LIN {X 0,Y 288.078,Z 352.641,A -85,B 0,C 180,E1 -18480.944,E2 -18480.944} C_VEL
LIN {X 0,Y 287.498,Z 347.512,A -85,B 0,C 180,E1 -18481.625,E2 -18481.625} C_VEL
LIN {X 0,Y 284.939,Z 340.607,A -85,B 0,C 180,E1 -18483.326,E2 -18483.326} C_VEL
LIN {X 0,Y 282.556,Z 335.313,A -85,B 0,C 180,E1 -18485.033,E2 -18485.033} C_VEL
LIN {X 0,Y 279.888,Z 329.784,A -85,B 0,C 180,E1 -18487.357,E2 -18487.357} C_VEL
LIN {X 0,Y 277.601,Z 325.434,A -85,B 0,C 180,E1 -18490.071,E2 -18490.071} C_VEL
LIN {X 0,Y 276.504,Z 323.001,A -85,B 0,C 180,E1 -18492.267,E2 -18492.267} C_VEL
LIN {X 0,Y 275.913,Z 321.671,A -85,B 0,C 180,E1 -18494.976,E2 -18494.976} C_VEL
LIN {X 0,Y 276.373,Z 321.734,A -85,B 0,C 180,E1 -18497.824,E2 -18497.824} C_VEL
LIN {X 0,Y 278.265,Z 323.737,A -85,B 0,C 180,E1 -18501.065,E2 -18501.065} C_VEL
LIN {X 0,Y 279.613,Z 325.391,A -85,B 0,C 180,E1 -18502.576,E2 -18502.576} C_VEL
LIN {X 0,Y 282.459,Z 329.547,A -85,B 0,C 180,E1 -18505.038,E2 -18505.038} C_VEL
LIN {X 0,Y 285.243,Z 334.015,A -85,B 0,C 180,E1 -18506.959,E2 -18506.959} C_VEL
LIN {X 0,Y 288.63,Z 340.16,A -85,B 0,C 180,E1 -18508.952,E2 -18508.952} C_VEL
LIN {X 0,Y 290.717,Z 344.56,A -85,B 0,C 180,E1 -18510.068,E2 -18510.068} C_VEL
LIN {X 0,Y 285.573,Z 380.843,A -85,B 0,C 180,E1 -18511.832,E2 -18511.832} C_VEL
LIN {X 0,Y 283.258,Z 392.365,A -85,B 0,C 180,E1 -18512.67,E2 -18512.67} C_VEL
LIN {X 0,Y 280.814,Z 402.262,A -85,B 0,C 180,E1 -18513.619,E2 -18513.619} C_VEL
LIN {X 0,Y 277.418,Z 413.784,A -85,B 0,C 180,E1 -18515.085,E2 -18515.085} C_VEL
LIN {X 0,Y 274.94,Z 421.064,A -85,B 0,C 180,E1 -18516.253,E2 -18516.253} C_VEL
LIN {X 0,Y 272.241,Z 428.033,A -85,B 0,C 180,E1 -18517.612,E2 -18517.612} C_VEL
LIN {X 0,Y 269.739,Z 433.852,A -85,B 0,C 180,E1 -18519,E2 -18519} C_VEL
LIN {X 0,Y 266.409,Z 441.005,A -85,B 0,C 180,E1 -18521.139,E2 -18521.139} C_VEL
LIN {X 0,Y 263.86,Z 445.653,A -85,B 0,C 180,E1 -18522.956,E2 -18522.956} C_VEL
LIN {X 0,Y 261.191,Z 449.803,A -85,B 0,C 180,E1 -18525.182,E2 -18525.182} C_VEL
LIN {X 0,Y 258.896,Z 452.702,A -85,B 0,C 180,E1 -18527.45,E2 -18527.45} C_VEL
LIN {X 0,Y 257.809,Z 453.984,A -85,B 0,C 180,E1 -18528.992,E2 -18528.992} C_VEL
LIN {X 0,Y 256.643,Z 454.794,A -85,B 0,C 180,E1 -18530.536,E2 -18530.536} C_VEL
LIN {X 0,Y 255.749,Z 454.994,A -85,B 0,C 180,E1 -18532.095,E2 -18532.095} C_VEL
LIN {X 0,Y 255.162,Z 454.673,A -85,B 0,C 180,E1 -18533.667,E2 -18533.667} C_VEL
LIN {X 0,Y 254.747,Z 453.89,A -85,B 0,C 180,E1 -18535.245,E2 -18535.245} C_VEL
LIN {X 0,Y 254.42,Z 452.619,A -85,B 0,C 180,E1 -18536.825,E2 -18536.825} C_VEL
LIN {X 0,Y 254.109,Z 449.575,A -85,B 0,C 180,E1 -18539.2,E2 -18539.2} C_VEL
LIN {X 0,Y 254.108,Z 445.253,A -85,B 0,C 180,E1 -18541.577,E2 -18541.577} C_VEL
LIN {X 0,Y 254.373,Z 439.511,A -85,B 0,C 180,E1 -18543.952,E2 -18543.952} C_VEL
LIN {X 0,Y 254.476,Z 433.189,A -85,B 0,C 180,E1 -18545.929,E2 -18545.929} C_VEL
LIN {X 0,Y 254.903,Z 425.839,A -85,B 0,C 180,E1 -18547.78,E2 -18547.78} C_VEL
LIN {X 0,Y 255.323,Z 417.479,A -85,B 0,C 180,E1 -18549.498,E2 -18549.498} C_VEL
LIN {X 0,Y 255.884,Z 406.564,A -85,B 0,C 180,E1 -18551.276,E2 -18551.276} C_VEL
LIN {X 0,Y 256.338,Z 397.268,A -85,B 0,C 180,E1 -18552.46,E2 -18552.46} C_VEL
LIN {X 0,Y 256.889,Z 386.565,A -85,B 0,C 180,E1 -18553.539,E2 -18553.539} C_VEL
LIN {X 0,Y 257.314,Z 373.603,A -85,B 0,C 180,E1 -18554.474,E2 -18554.474} C_VEL
LIN {X 0,Y 258.64,Z 317.417,A -85,B 0,C 180,E1 -18557.079,E2 -18557.079} C_VEL
LIN {X 0,Y 256.336,Z 296.461,A -85,B 0,C 180,E1 -18558.059,E2 -18558.059} C_VEL
LIN {X 0,Y 256.227,Z 294.598,A -85,B 0,C 180,E1 -18558.171,E2 -18558.171} C_VEL
LIN {X 0,Y 256.274,Z 293.374,A -85,B 0,C 180,E1 -18558.788,E2 -18558.788} C_VEL
LIN {X 0,Y 256.19,Z 293.381,A -85,B 0,C 180,E1 -18561.133,E2 -18561.133} C_VEL
LIN {X 0,Y 256.054,Z 293.402,A -85,B 0,C 180,E1 -18566.04,E2 -18566.04} C_VEL
LIN {X 0,Y 256.026,Z 293.403,A -85,B 0,C 180,E1 -18569.6,E2 -18569.6} C_VEL
LIN {X 0,Y 256.048,Z 293.399,A -85,B 0,C 180,E1 -18573.284,E2 -18573.284} C_VEL
LIN {X 0,Y 256.066,Z 293.398,A -85,B 0,C 180,E1 -18577.253,E2 -18577.253} C_VEL
LIN {X 0,Y 255.984,Z 293.408,A -85,B 0,C 180,E1 -18581.204,E2 -18581.204} C_VEL
LIN {X 0,Y 256.009,Z 293.405,A -85,B 0,C 180,E1 -18585.527,E2 -18585.527} C_VEL
LIN {X 0,Y 256.021,Z 293.406,A -85,B 0,C 180,E1 -18588.787,E2 -18588.787} C_VEL
LIN {X 0,Y 256.097,Z 293.398,A -85,B 0,C 180,E1 -18592.859,E2 -18592.859} C_VEL
LIN {X 0,Y 256.031,Z 293.404,A -85,B 0,C 180,E1 -18596.699,E2 -18596.699} C_VEL
LIN {X 0,Y 256.028,Z 293.402,A -85,B 0,C 180,E1 -18600.387,E2 -18600.387} C_VEL
LIN {X 0,Y 256.088,Z 293.396,A -85,B 0,C 180,E1 -18603.951,E2 -18603.951} C_VEL
LIN {X 0,Y 256.041,Z 293.403,A -85,B 0,C 180,E1 -18607.398,E2 -18607.398} C_VEL
LIN {X 0,Y 256.14,Z 293.389,A -85,B 0,C 180,E1 -18610.774,E2 -18610.774} C_VEL
LIN {X 0,Y 256.22,Z 293.379,A -85,B 0,C 180,E1 -18614.077,E2 -18614.077} C_VEL
LIN {X 0,Y 256.262,Z 293.373,A -85,B 0,C 180,E1 -18618.929,E2 -18618.929} C_VEL
LIN {X 0,Y 256.482,Z 293.348,A -85,B 0,C 180,E1 -18622.123,E2 -18622.123} C_VEL
LIN {X 0,Y 256.672,Z 293.324,A -85,B 0,C 180,E1 -18628.428,E2 -18628.428} C_VEL
LIN {X 0,Y 256.671,Z 293.324,A -85,B 0,C 180,E1 -18631.566,E2 -18631.566} C_VEL
LIN {X 0,Y 256.478,Z 293.349,A -85,B 0,C 180,E1 -18637.872,E2 -18637.872} C_VEL
LIN {X 0,Y 256.258,Z 293.374,A -85,B 0,C 180,E1 -18641.065,E2 -18641.065} C_VEL
LIN {X 0,Y 256.213,Z 293.38,A -85,B 0,C 180,E1 -18645.917,E2 -18645.917} C_VEL
LIN {X 0,Y 256.132,Z 293.39,A -85,B 0,C 180,E1 -18649.221,E2 -18649.221} C_VEL
LIN {X 0,Y 256.032,Z 293.404,A -85,B 0,C 180,E1 -18652.597,E2 -18652.597} C_VEL
LIN {X 0,Y 256.079,Z 293.397,A -85,B 0,C 180,E1 -18656.044,E2 -18656.044} C_VEL
LIN {X 0,Y 256.065,Z 293.397,A -85,B 0,C 180,E1 -18659.602,E2 -18659.602} C_VEL
LIN {X 0,Y 256.038,Z 293.403,A -85,B 0,C 180,E1 -18663.293,E2 -18663.293} C_VEL
LIN {X 0,Y 256.093,Z 293.397,A -85,B 0,C 180,E1 -18667.282,E2 -18667.282} C_VEL
LIN {X 0,Y 256.088,Z 293.398,A -85,B 0,C 180,E1 -18671.193,E2 -18671.193} C_VEL
LIN {X 0,Y 256.074,Z 293.4,A -85,B 0,C 180,E1 -18675.522,E2 -18675.522} C_VEL
LIN {X 0,Y 256.091,Z 293.395,A -85,B 0,C 180,E1 -18678.817,E2 -18678.817} C_VEL
LIN {X 0,Y 256.115,Z 293.392,A -85,B 0,C 180,E1 -18682.877,E2 -18682.877} C_VEL
LIN {X 0,Y 256.049,Z 293.399,A -85,B 0,C 180,E1 -18686.716,E2 -18686.716} C_VEL
LIN {X 0,Y 256.093,Z 293.397,A -85,B 0,C 180,E1 -18691.417,E2 -18691.417} C_VEL
LIN {X 0,Y 256.111,Z 293.396,A -85,B 0,C 180,E1 -18695.704,E2 -18695.704} C_VEL
LIN {X 0,Y 256.119,Z 293.39,A -85,B 0,C 180,E1 -18699.111,E2 -18699.111} C_VEL
LIN {X 0,Y 256.22,Z 293.382,A -85,B 0,C 180,E1 -18704.089,E2 -18704.089} C_VEL
LIN {X 0,Y 256.268,Z 293.373,A -85,B 0,C 180,E1 -18708.941,E2 -18708.941} C_VEL
LIN {X 0,Y 256.478,Z 293.351,A -85,B 0,C 180,E1 -18712.134,E2 -18712.134} C_VEL
LIN {X 0,Y 256.439,Z 293.352,A -85,B 0,C 180,E1 -18716.866,E2 -18716.866} C_VEL
LIN {X 0,Y 256.686,Z 293.325,A -85,B 0,C 180,E1 -18718.439,E2 -18718.439} C_VEL
LIN {X 0,Y 256.686,Z 293.321,A -85,B 0,C 180,E1 -18721.577,E2 -18721.577} C_VEL
LIN {X 0,Y 256.445,Z 293.351,A -85,B 0,C 180,E1 -18726.301,E2 -18726.301} C_VEL
LIN {X 0,Y 256.393,Z 293.358,A -85,B 0,C 180,E1 -18729.474,E2 -18729.474} C_VEL
LIN {X 0,Y 256.198,Z 293.38,A -85,B 0,C 180,E1 -18734.301,E2 -18734.301} C_VEL
LIN {X 0,Y 256.142,Z 293.389,A -85,B 0,C 180,E1 -18737.574,E2 -18737.574} C_VEL
LIN {X 0,Y 256.115,Z 293.395,A -85,B 0,C 180,E1 -18741.104,E2 -18741.104} C_VEL
LIN {X 0,Y 256.083,Z 293.399,A -85,B 0,C 180,E1 -18745.096,E2 -18745.096} C_VEL
LIN {X 0,Y 256.086,Z 293.396,A -85,B 0,C 180,E1 -18748.581,E2 -18748.581} C_VEL
LIN {X 0,Y 256.075,Z 293.398,A -85,B 0,C 180,E1 -18751.708,E2 -18751.708} C_VEL
LIN {X 0,Y 256.066,Z 293.399,A -85,B 0,C 180,E1 -18753.482,E2 -18753.482} C_VEL
LIN {X 0,Y 255.413,Z 293.481,A -85,B 0,C 180,E1 -18754.795,E2 -18754.795} C_VEL
LIN {X 0,Y 252.605,Z 293.833,A -85,B 0,C 180,E1 -18756.938,E2 -18756.938} C_VEL
LIN {X 0,Y 249.35,Z 294.238,A -85,B 0,C 180,E1 -18759.577,E2 -18759.577} C_VEL
LIN {X 0,Y 248.983,Z 294.278,A -85,B 0,C 180,E1 -18760.491,E2 -18760.491} C_VEL
LIN {X 0,Y 248.968,Z 294.282,A -85,B 0,C 180,E1 -18764.895,E2 -18764.895} C_VEL
LIN {X 0,Y 248.986,Z 294.281,A -85,B 0,C 180,E1 -18767.361,E2 -18767.361} C_VEL
LIN {X 0,Y 249.053,Z 294.274,A -85,B 0,C 180,E1 -18772.207,E2 -18772.207} C_VEL
LIN {X 0,Y 249.053,Z 294.273,A -85,B 0,C 180,E1 -18775.645,E2 -18775.645} C_VEL
LIN {X 0,Y 249.01,Z 294.275,A -85,B 0,C 180,E1 -18779.471,E2 -18779.471} C_VEL
LIN {X 0,Y 249.328,Z 294.267,A -85,B 0,C 180,E1 -18783.991,E2 -18783.991} C_VEL
LIN {X 0,Y 250.346,Z 300.279,A -85,B 0,C 180,E1 -18786.423,E2 -18786.423} C_VEL
LIN {X 0,Y 249.092,Z 310.954,A -85,B 0,C 180,E1 -18790.642,E2 -18790.642} C_VEL
LIN {X 0,Y 248.799,Z 313.594,A -85,B 0,C 180,E1 -18791.687,E2 -18791.687} C_VEL
LIN {X 0,Y 249.482,Z 331.264,A -85,B 0,C 180,E1 -18792.554,E2 -18792.554} C_VEL
LIN {X 0,Y 251.209,Z 351.622,A -85,B 0,C 180,E1 -18793.536,E2 -18793.536} C_VEL
LIN {X 0,Y 250.2,Z 393.642,A -85,B 0,C 180,E1 -18795.619,E2 -18795.619} C_VEL
LIN {X 0,Y 249.777,Z 405.976,A -85,B 0,C 180,E1 -18796.58,E2 -18796.58} C_VEL
LIN {X 0,Y 249.294,Z 415.542,A -85,B 0,C 180,E1 -18797.59,E2 -18797.59} C_VEL
LIN {X 0,Y 248.756,Z 426.15,A -85,B 0,C 180,E1 -18799.009,E2 -18799.009} C_VEL
LIN {X 0,Y 248.379,Z 435.573,A -85,B 0,C 180,E1 -18800.639,E2 -18800.639} C_VEL
LIN {X 0,Y 248.049,Z 443.217,A -85,B 0,C 180,E1 -18802.274,E2 -18802.274} C_VEL
LIN {X 0,Y 247.91,Z 449.562,A -85,B 0,C 180,E1 -18803.91,E2 -18803.91} C_VEL
LIN {X 0,Y 247.768,Z 454.731,A -85,B 0,C 180,E1 -18805.529,E2 -18805.529} C_VEL
LIN {X 0,Y 247.6,Z 459.948,A -85,B 0,C 180,E1 -18807.563,E2 -18807.563} C_VEL
LIN {X 0,Y 247.634,Z 464.762,A -85,B 0,C 180,E1 -18810.003,E2 -18810.003} C_VEL
LIN {X 0,Y 247.206,Z 466.989,A -85,B 0,C 180,E1 -18811.632,E2 -18811.632} C_VEL
LIN {X 0,Y 247.115,Z 468.697,A -85,B 0,C 180,E1 -18813.263,E2 -18813.263} C_VEL
LIN {X 0,Y 247.11,Z 470.165,A -85,B 0,C 180,E1 -18815.429,E2 -18815.429} C_VEL
LIN {X 0,Y 247.201,Z 470.623,A -85,B 0,C 180,E1 -18816.533,E2 -18816.533} C_VEL
LIN {X 0,Y 247.539,Z 470.786,A -85,B 0,C 180,E1 -18818.164,E2 -18818.164} C_VEL
LIN {X 0,Y 248.096,Z 470.422,A -85,B 0,C 180,E1 -18819.789,E2 -18819.789} C_VEL
LIN {X 0,Y 248.913,Z 469.615,A -85,B 0,C 180,E1 -18821.402,E2 -18821.402} C_VEL
LIN {X 0,Y 249.993,Z 468.35,A -85,B 0,C 180,E1 -18823,E2 -18823} C_VEL
LIN {X 0,Y 252.028,Z 465.39,A -85,B 0,C 180,E1 -18825.364,E2 -18825.364} C_VEL
LIN {X 0,Y 253.723,Z 462.798,A -85,B 0,C 180,E1 -18826.911,E2 -18826.911} C_VEL
LIN {X 0,Y 256.501,Z 457.656,A -85,B 0,C 180,E1 -18829.198,E2 -18829.198} C_VEL
LIN {X 0,Y 259.354,Z 452.305,A -85,B 0,C 180,E1 -18831.044,E2 -18831.044} C_VEL
LIN {X 0,Y 262.607,Z 445.702,A -85,B 0,C 180,E1 -18832.836,E2 -18832.836} C_VEL
LIN {X 0,Y 266.26,Z 437.594,A -85,B 0,C 180,E1 -18834.567,E2 -18834.567} C_VEL
LIN {X 0,Y 269.842,Z 428.59,A -85,B 0,C 180,E1 -18836.075,E2 -18836.075} C_VEL
LIN {X 0,Y 272.91,Z 420.038,A -85,B 0,C 180,E1 -18837.202,E2 -18837.202} C_VEL
LIN {X 0,Y 275.659,Z 411.201,A -85,B 0,C 180,E1 -18838.145,E2 -18838.145} C_VEL
LIN {X 0,Y 278.901,Z 399.082,A -85,B 0,C 180,E1 -18839.123,E2 -18839.123} C_VEL
LIN {X 0,Y 281.328,Z 386.651,A -85,B 0,C 180,E1 -18839.875,E2 -18839.875} C_VEL
LIN {X 0,Y 284.531,Z 364.834,A -85,B 0,C 180,E1 -18840.937,E2 -18840.937} C_VEL
LIN {X 0,Y 284.092,Z 354.378,A -85,B 0,C 180,E1 -18842.129,E2 -18842.129} C_VEL
LIN {X 0,Y 283.77,Z 351.646,A -85,B 0,C 180,E1 -18842.551,E2 -18842.551} C_VEL
LIN {X 0,Y 281.525,Z 345.515,A -85,B 0,C 180,E1 -18844.168,E2 -18844.168} C_VEL
LIN {X 0,Y 279.677,Z 341.044,A -85,B 0,C 180,E1 -18845.691,E2 -18845.691} C_VEL
LIN {X 0,Y 277.489,Z 336.114,A -85,B 0,C 180,E1 -18847.818,E2 -18847.818} C_VEL
LIN {X 0,Y 275.344,Z 331.685,A -85,B 0,C 180,E1 -18850.66,E2 -18850.66} C_VEL
LIN {X 0,Y 274.535,Z 329.607,A -85,B 0,C 180,E1 -18852.644,E2 -18852.644} C_VEL
LIN {X 0,Y 274.11,Z 328.543,A -85,B 0,C 180,E1 -18854.977,E2 -18854.977} C_VEL
LIN {X 0,Y 274.456,Z 328.463,A -85,B 0,C 180,E1 -18857.484,E2 -18857.484} C_VEL
LIN {X 0,Y 276.365,Z 330.545,A -85,B 0,C 180,E1 -18860.979,E2 -18860.979} C_VEL
LIN {X 0,Y 277.561,Z 332.177,A -85,B 0,C 180,E1 -18862.414,E2 -18862.414} C_VEL
LIN {X 0,Y 279.95,Z 335.855,A -85,B 0,C 180,E1 -18864.624,E2 -18864.624} C_VEL
LIN {X 0,Y 282.575,Z 340.41,A -85,B 0,C 180,E1 -18866.592,E2 -18866.592} C_VEL
LIN {X 0,Y 285.617,Z 346.256,A -85,B 0,C 180,E1 -18868.504,E2 -18868.504} C_VEL
LIN {X 0,Y 286.579,Z 348.295,A -85,B 0,C 180,E1 -18869.052,E2 -18869.052} C_VEL
LIN {X 0,Y 281.589,Z 380.533,A -85,B 0,C 180,E1 -18870.614,E2 -18870.614} C_VEL
LIN {X 0,Y 279.233,Z 391.744,A -85,B 0,C 180,E1 -18871.425,E2 -18871.425} C_VEL
LIN {X 0,Y 276.604,Z 401.83,A -85,B 0,C 180,E1 -18872.367,E2 -18872.367} C_VEL
LIN {X 0,Y 273.406,Z 412.453,A -85,B 0,C 180,E1 -18873.671,E2 -18873.671} C_VEL
LIN {X 0,Y 270.319,Z 420.838,A -85,B 0,C 180,E1 -18875.002,E2 -18875.002} C_VEL
LIN {X 0,Y 266.726,Z 429.403,A -85,B 0,C 180,E1 -18876.712,E2 -18876.712} C_VEL
LIN {X 0,Y 263.432,Z 436.434,A -85,B 0,C 180,E1 -18878.473,E2 -18878.473} C_VEL
LIN {X 0,Y 260.508,Z 442,A -85,B 0,C 180,E1 -18880.285,E2 -18880.285} C_VEL
LIN {X 0,Y 257.237,Z 447.173,A -85,B 0,C 180,E1 -18882.503,E2 -18882.503} C_VEL
LIN {X 0,Y 254.456,Z 451.035,A -85,B 0,C 180,E1 -18884.781,E2 -18884.781} C_VEL
LIN {X 0,Y 253.559,Z 452.117,A -85,B 0,C 180,E1 -18885.547,E2 -18885.547} C_VEL
LIN {X 0,Y 252.043,Z 453.653,A -85,B 0,C 180,E1 -18887.103,E2 -18887.103} C_VEL
LIN {X 0,Y 250.885,Z 454.66,A -85,B 0,C 180,E1 -18888.684,E2 -18888.684} C_VEL
LIN {X 0,Y 249.669,Z 455.239,A -85,B 0,C 180,E1 -18890.269,E2 -18890.269} C_VEL
LIN {X 0,Y 248.732,Z 455.338,A -85,B 0,C 180,E1 -18891.871,E2 -18891.871} C_VEL
LIN {X 0,Y 248.107,Z 454.848,A -85,B 0,C 180,E1 -18893.486,E2 -18893.486} C_VEL
LIN {X 0,Y 247.682,Z 453.826,A -85,B 0,C 180,E1 -18895.109,E2 -18895.109} C_VEL
LIN {X 0,Y 247.211,Z 451.421,A -85,B 0,C 180,E1 -18897.548,E2 -18897.548} C_VEL
LIN {X 0,Y 247.02,Z 447.737,A -85,B 0,C 180,E1 -18899.992,E2 -18899.992} C_VEL
LIN {X 0,Y 247.135,Z 442.542,A -85,B 0,C 180,E1 -18902.436,E2 -18902.436} C_VEL
LIN {X 0,Y 247.322,Z 438.239,A -85,B 0,C 180,E1 -18904.065,E2 -18904.065} C_VEL
LIN {X 0,Y 247.471,Z 431.905,A -85,B 0,C 180,E1 -18906.014,E2 -18906.014} C_VEL
LIN {X 0,Y 247.853,Z 425.134,A -85,B 0,C 180,E1 -18907.732,E2 -18907.732} C_VEL
LIN {X 0,Y 248.308,Z 416.296,A -85,B 0,C 180,E1 -18909.563,E2 -18909.563} C_VEL
LIN {X 0,Y 248.805,Z 406.247,A -85,B 0,C 180,E1 -18911.189,E2 -18911.189} C_VEL
LIN {X 0,Y 249.261,Z 396.831,A -85,B 0,C 180,E1 -18912.406,E2 -18912.406} C_VEL
LIN {X 0,Y 249.824,Z 385.992,A -85,B 0,C 180,E1 -18913.514,E2 -18913.514} C_VEL
LIN {X 0,Y 250.222,Z 373.37,A -85,B 0,C 180,E1 -18914.425,E2 -18914.425} C_VEL
LIN {X 0,Y 251.46,Z 317.095,A -85,B 0,C 180,E1 -18917.152,E2 -18917.152} C_VEL
LIN {X 0,Y 249.248,Z 296.678,A -85,B 0,C 180,E1 -18918.139,E2 -18918.139} C_VEL
LIN {X 0,Y 249.146,Z 294.806,A -85,B 0,C 180,E1 -18918.28,E2 -18918.28} C_VEL
LIN {X 0,Y 249.181,Z 294.258,A -85,B 0,C 180,E1 -18918.597,E2 -18918.597} C_VEL
LIN {X 0,Y 249.097,Z 294.266,A -85,B 0,C 180,E1 -18921.507,E2 -18921.507} C_VEL
LIN {X 0,Y 249.033,Z 294.274,A -85,B 0,C 180,E1 -18925.43,E2 -18925.43} C_VEL
LIN {X 0,Y 249.01,Z 294.277,A -85,B 0,C 180,E1 -18928.958,E2 -18928.958} C_VEL
LIN {X 0,Y 249.009,Z 294.279,A -85,B 0,C 180,E1 -18932.417,E2 -18932.417} C_VEL
LIN {X 0,Y 248.991,Z 294.283,A -85,B 0,C 180,E1 -18936.339,E2 -18936.339} C_VEL
LIN {X 0,Y 248.949,Z 294.286,A -85,B 0,C 180,E1 -18940.476,E2 -18940.476} C_VEL
LIN {X 0,Y 248.948,Z 294.288,A -85,B 0,C 180,E1 -18944.877,E2 -18944.877} C_VEL
LIN {X 0,Y 248.978,Z 294.281,A -85,B 0,C 180,E1 -18947.352,E2 -18947.352} C_VEL
LIN {X 0,Y 249.011,Z 294.277,A -85,B 0,C 180,E1 -18952.192,E2 -18952.192} C_VEL
LIN {X 0,Y 249.009,Z 294.277,A -85,B 0,C 180,E1 -18955.631,E2 -18955.631} C_VEL
LIN {X 0,Y 248.97,Z 294.283,A -85,B 0,C 180,E1 -18959.459,E2 -18959.459} C_VEL
LIN {X 0,Y 249.024,Z 294.279,A -85,B 0,C 180,E1 -18963.154,E2 -18963.154} C_VEL
LIN {X 0,Y 249.019,Z 294.275,A -85,B 0,C 180,E1 -18966.724,E2 -18966.724} C_VEL
LIN {X 0,Y 249.064,Z 294.27,A -85,B 0,C 180,E1 -18970.205,E2 -18970.205} C_VEL
LIN {X 0,Y 249.152,Z 294.263,A -85,B 0,C 180,E1 -18973.613,E2 -18973.613} C_VEL
LIN {X 0,Y 249.205,Z 294.252,A -85,B 0,C 180,E1 -18978.612,E2 -18978.612} C_VEL
LIN {X 0,Y 249.423,Z 294.229,A -85,B 0,C 180,E1 -18981.898,E2 -18981.898} C_VEL
LIN {X 0,Y 249.416,Z 294.225,A -85,B 0,C 180,E1 -18986.767,E2 -18986.767} C_VEL
LIN {X 0,Y 249.685,Z 294.198,A -85,B 0,C 180,E1 -18989.997,E2 -18989.997} C_VEL
LIN {X 0,Y 249.414,Z 294.225,A -85,B 0,C 180,E1 -18993.228,E2 -18993.228} C_VEL
LIN {X 0,Y 249.419,Z 294.229,A -85,B 0,C 180,E1 -18998.096,E2 -18998.096} C_VEL
LIN {X 0,Y 249.2,Z 294.253,A -85,B 0,C 180,E1 -19001.383,E2 -19001.383} C_VEL
LIN {X 0,Y 249.146,Z 294.264,A -85,B 0,C 180,E1 -19006.486,E2 -19006.486} C_VEL
LIN {X 0,Y 249.043,Z 294.271,A -85,B 0,C 180,E1 -19011.399,E2 -19011.399} C_VEL
LIN {X 0,Y 249.067,Z 294.27,A -85,B 0,C 180,E1 -19015.477,E2 -19015.477} C_VEL
LIN {X 0,Y 249.034,Z 294.276,A -85,B 0,C 180,E1 -19018.995,E2 -19018.995} C_VEL
LIN {X 0,Y 248.988,Z 294.279,A -85,B 0,C 180,E1 -19022.428,E2 -19022.428} C_VEL
LIN {X 0,Y 249.028,Z 294.275,A -85,B 0,C 180,E1 -19026.342,E2 -19026.342} C_VEL
LIN {X 0,Y 249.039,Z 294.271,A -85,B 0,C 180,E1 -19030.467,E2 -19030.467} C_VEL
LIN {X 0,Y 249.05,Z 294.273,A -85,B 0,C 180,E1 -19032.818,E2 -19032.818} C_VEL
LIN {X 0,Y 249.057,Z 294.274,A -85,B 0,C 180,E1 -19037.385,E2 -19037.385} C_VEL
LIN {X 0,Y 249.013,Z 294.28,A -85,B 0,C 180,E1 -19041.63,E2 -19041.63} C_VEL
LIN {X 0,Y 249.025,Z 294.278,A -85,B 0,C 180,E1 -19045.649,E2 -19045.649} C_VEL
LIN {X 0,Y 249.013,Z 294.277,A -85,B 0,C 180,E1 -19049.479,E2 -19049.479} C_VEL
LIN {X 0,Y 249.036,Z 294.275,A -85,B 0,C 180,E1 -19053.169,E2 -19053.169} C_VEL
LIN {X 0,Y 249.03,Z 294.272,A -85,B 0,C 180,E1 -19056.738,E2 -19056.738} C_VEL
LIN {X 0,Y 249.054,Z 294.274,A -85,B 0,C 180,E1 -19060.217,E2 -19060.217} C_VEL
LIN {X 0,Y 249.17,Z 294.259,A -85,B 0,C 180,E1 -19063.626,E2 -19063.626} C_VEL
LIN {X 0,Y 249.211,Z 294.253,A -85,B 0,C 180,E1 -19068.624,E2 -19068.624} C_VEL
LIN {X 0,Y 249.421,Z 294.228,A -85,B 0,C 180,E1 -19071.91,E2 -19071.91} C_VEL
LIN {X 0,Y 249.253,Z 294.244,A -85,B 0,C 180,E1 -19075.156,E2 -19075.156} C_VEL
LIN {X 0,Y 249.646,Z 294.201,A -85,B 0,C 180,E1 -19078.395,E2 -19078.395} C_VEL
LIN {X 0,Y 249.647,Z 294.197,A -85,B 0,C 180,E1 -19081.621,E2 -19081.621} C_VEL
LIN {X 0,Y 249.416,Z 294.228,A -85,B 0,C 180,E1 -19086.479,E2 -19086.479} C_VEL
LIN {X 0,Y 249.324,Z 294.238,A -85,B 0,C 180,E1 -19089.745,E2 -19089.745} C_VEL
LIN {X 0,Y 249.142,Z 294.261,A -85,B 0,C 180,E1 -19094.715,E2 -19094.715} C_VEL
LIN {X 0,Y 249.074,Z 294.269,A -85,B 0,C 180,E1 -19098.09,E2 -19098.09} C_VEL
LIN {X 0,Y 249.039,Z 294.272,A -85,B 0,C 180,E1 -19101.53,E2 -19101.53} C_VEL
LIN {X 0,Y 249.045,Z 294.276,A -85,B 0,C 180,E1 -19105.448,E2 -19105.448} C_VEL
LIN {X 0,Y 249.034,Z 294.276,A -85,B 0,C 180,E1 -19108.98,E2 -19108.98} C_VEL
LIN {X 0,Y 249.003,Z 294.273,A -85,B 0,C 180,E1 -19113.487,E2 -19113.487} C_VEL
LIN {X 0,Y 249.047,Z 294.274,A -85,B 0,C 180,E1 -19117.806,E2 -19117.806} C_VEL
LIN {X 0,Y 248.983,Z 294.278,A -85,B 0,C 180,E1 -19120.491,E2 -19120.491} C_VEL
LIN {X 0,Y 248.239,Z 294.376,A -85,B 0,C 180,E1 -19121.84,E2 -19121.84} C_VEL
LIN {X 0,Y 245.348,Z 294.736,A -85,B 0,C 180,E1 -19124.04,E2 -19124.04} C_VEL
LIN {X 0,Y 242.957,Z 295.035,A -85,B 0,C 180,E1 -19125.832,E2 -19125.832} C_VEL
LIN {X 0,Y 241.963,Z 295.155,A -85,B 0,C 180,E1 -19127.221,E2 -19127.221} C_VEL
LIN {X 0,Y 241.897,Z 295.161,A -85,B 0,C 180,E1 -19127.692,E2 -19127.692} C_VEL
LIN {X 0,Y 242.003,Z 295.151,A -85,B 0,C 180,E1 -19131.648,E2 -19131.648} C_VEL
LIN {X 0,Y 241.984,Z 295.154,A -85,B 0,C 180,E1 -19134.493,E2 -19134.493} C_VEL
LIN {X 0,Y 241.961,Z 295.155,A -85,B 0,C 180,E1 -19138.482,E2 -19138.482} C_VEL
LIN {X 0,Y 242.307,Z 295.12,A -85,B 0,C 180,E1 -19144.135,E2 -19144.135} C_VEL
LIN {X 0,Y 243.237,Z 299.948,A -85,B 0,C 180,E1 -19146.143,E2 -19146.143} C_VEL
LIN {X 0,Y 242.392,Z 307.442,A -85,B 0,C 180,E1 -19149.199,E2 -19149.199} C_VEL
LIN {X 0,Y 241.726,Z 313.336,A -85,B 0,C 180,E1 -19151.613,E2 -19151.613} C_VEL
LIN {X 0,Y 242.353,Z 331.256,A -85,B 0,C 180,E1 -19152.547,E2 -19152.547} C_VEL
LIN {X 0,Y 244.114,Z 351.259,A -85,B 0,C 180,E1 -19153.54,E2 -19153.54} C_VEL
LIN {X 0,Y 243.141,Z 392.775,A -85,B 0,C 180,E1 -19155.674,E2 -19155.674} C_VEL
LIN {X 0,Y 242.754,Z 404.796,A -85,B 0,C 180,E1 -19156.611,E2 -19156.611} C_VEL
LIN {X 0,Y 242.266,Z 414.505,A -85,B 0,C 180,E1 -19157.649,E2 -19157.649} C_VEL
LIN {X 0,Y 241.751,Z 423.785,A -85,B 0,C 180,E1 -19158.899,E2 -19158.899} C_VEL
LIN {X 0,Y 241.379,Z 433.74,A -85,B 0,C 180,E1 -19160.577,E2 -19160.577} C_VEL
LIN {X 0,Y 241.053,Z 442.428,A -85,B 0,C 180,E1 -19162.468,E2 -19162.468} C_VEL
LIN {X 0,Y 240.915,Z 448.756,A -85,B 0,C 180,E1 -19164.143,E2 -19164.143} C_VEL
LIN {X 0,Y 240.793,Z 454.006,A -85,B 0,C 180,E1 -19165.818,E2 -19165.818} C_VEL
LIN {X 0,Y 240.648,Z 458.337,A -85,B 0,C 180,E1 -19167.492,E2 -19167.492} C_VEL
LIN {X 0,Y 240.634,Z 463.434,A -85,B 0,C 180,E1 -19170.003,E2 -19170.003} C_VEL
LIN {X 0,Y 240.222,Z 465.893,A -85,B 0,C 180,E1 -19171.679,E2 -19171.679} C_VEL
LIN {X 0,Y 240.089,Z 467.804,A -85,B 0,C 180,E1 -19173.359,E2 -19173.359} C_VEL
LIN {X 0,Y 240.049,Z 469.411,A -85,B 0,C 180,E1 -19175.427,E2 -19175.427} C_VEL
LIN {X 0,Y 240.172,Z 470.036,A -85,B 0,C 180,E1 -19176.725,E2 -19176.725} C_VEL
LIN {X 0,Y 240.504,Z 470.359,A -85,B 0,C 180,E1 -19178.404,E2 -19178.404} C_VEL
LIN {X 0,Y 241.088,Z 470.245,A -85,B 0,C 180,E1 -19180.076,E2 -19180.076} C_VEL
LIN {X 0,Y 241.972,Z 469.687,A -85,B 0,C 180,E1 -19181.733,E2 -19181.733} C_VEL
LIN {X 0,Y 243.09,Z 468.545,A -85,B 0,C 180,E1 -19183.376,E2 -19183.376} C_VEL
LIN {X 0,Y 245.231,Z 465.97,A -85,B 0,C 180,E1 -19185.801,E2 -19185.801} C_VEL
LIN {X 0,Y 247.838,Z 462.169,A -85,B 0,C 180,E1 -19188.178,E2 -19188.178} C_VEL
LIN {X 0,Y 251.058,Z 457.016,A -85,B 0,C 180,E1 -19190.485,E2 -19190.485} C_VEL
LIN {X 0,Y 254.221,Z 451.554,A -85,B 0,C 180,E1 -19192.344,E2 -19192.344} C_VEL
LIN {X 0,Y 258.511,Z 443.506,A -85,B 0,C 180,E1 -19194.496,E2 -19194.496} C_VEL
LIN {X 0,Y 262.434,Z 434.979,A -85,B 0,C 180,E1 -19196.226,E2 -19196.226} C_VEL
LIN {X 0,Y 265.914,Z 426.584,A -85,B 0,C 180,E1 -19197.552,E2 -19197.552} C_VEL
LIN {X 0,Y 270.215,Z 415.054,A -85,B 0,C 180,E1 -19198.977,E2 -19198.977} C_VEL
LIN {X 0,Y 273.761,Z 403.269,A -85,B 0,C 180,E1 -19200.042,E2 -19200.042} C_VEL
LIN {X 0,Y 276.694,Z 391.182,A -85,B 0,C 180,E1 -19200.865,E2 -19200.865} C_VEL
LIN {X 0,Y 280.644,Z 366.61,A -85,B 0,C 180,E1 -19202.103,E2 -19202.103} C_VEL
LIN {X 0,Y 280.416,Z 356.731,A -85,B 0,C 180,E1 -19203.308,E2 -19203.308} C_VEL
LIN {X 0,Y 278.66,Z 351.339,A -85,B 0,C 180,E1 -19204.766,E2 -19204.766} C_VEL
LIN {X 0,Y 276.922,Z 346.906,A -85,B 0,C 180,E1 -19206.292,E2 -19206.292} C_VEL
LIN {X 0,Y 275.063,Z 342.303,A -85,B 0,C 180,E1 -19208.335,E2 -19208.335} C_VEL
LIN {X 0,Y 273.213,Z 337.983,A -85,B 0,C 180,E1 -19211.259,E2 -19211.259} C_VEL
LIN {X 0,Y 272.536,Z 336.138,A -85,B 0,C 180,E1 -19213.207,E2 -19213.207} C_VEL
LIN {X 0,Y 272.333,Z 335.299,A -85,B 0,C 180,E1 -19215.824,E2 -19215.824} C_VEL
LIN {X 0,Y 272.8,Z 335.517,A -85,B 0,C 180,E1 -19217.939,E2 -19217.939} C_VEL
LIN {X 0,Y 274.752,Z 337.684,A -85,B 0,C 180,E1 -19221.267,E2 -19221.267} C_VEL
LIN {X 0,Y 277.509,Z 342.235,A -85,B 0,C 180,E1 -19224.232,E2 -19224.232} C_VEL
LIN {X 0,Y 280.17,Z 347.088,A -85,B 0,C 180,E1 -19226.337,E2 -19226.337} C_VEL
LIN {X 0,Y 282.552,Z 352.005,A -85,B 0,C 180,E1 -19227.941,E2 -19227.941} C_VEL
LIN {X 0,Y 277.687,Z 381.418,A -85,B 0,C 180,E1 -19229.417,E2 -19229.417} C_VEL
LIN {X 0,Y 274.963,Z 393.467,A -85,B 0,C 180,E1 -19230.308,E2 -19230.308} C_VEL
LIN {X 0,Y 272.188,Z 403.218,A -85,B 0,C 180,E1 -19231.249,E2 -19231.249} C_VEL
LIN {X 0,Y 268.323,Z 414.525,A -85,B 0,C 180,E1 -19232.712,E2 -19232.712} C_VEL
LIN {X 0,Y 265.092,Z 422.644,A -85,B 0,C 180,E1 -19234.052,E2 -19234.052} C_VEL
LIN {X 0,Y 262.048,Z 429.417,A -85,B 0,C 180,E1 -19235.429,E2 -19235.429} C_VEL
LIN {X 0,Y 258.469,Z 436.418,A -85,B 0,C 180,E1 -19237.196,E2 -19237.196} C_VEL
LIN {X 0,Y 255.273,Z 442.065,A -85,B 0,C 180,E1 -19239.021,E2 -19239.021} C_VEL
LIN {X 0,Y 251.716,Z 447.335,A -85,B 0,C 180,E1 -19241.264,E2 -19241.264} C_VEL
LIN {X 0,Y 248.638,Z 451.202,A -85,B 0,C 180,E1 -19243.573,E2 -19243.573} C_VEL
LIN {X 0,Y 246.785,Z 453.119,A -85,B 0,C 180,E1 -19245.142,E2 -19245.142} C_VEL
LIN {X 0,Y 245.2,Z 454.545,A -85,B 0,C 180,E1 -19246.736,E2 -19246.736} C_VEL
LIN {X 0,Y 243.978,Z 455.367,A -85,B 0,C 180,E1 -19248.359,E2 -19248.359} C_VEL
LIN {X 0,Y 242.697,Z 455.675,A -85,B 0,C 180,E1 -19249.986,E2 -19249.986} C_VEL
LIN {X 0,Y 241.711,Z 455.518,A -85,B 0,C 180,E1 -19251.633,E2 -19251.633} C_VEL
LIN {X 0,Y 241.058,Z 454.905,A -85,B 0,C 180,E1 -19253.295,E2 -19253.295} C_VEL
LIN {X 0,Y 240.622,Z 453.741,A -85,B 0,C 180,E1 -19254.965,E2 -19254.965} C_VEL
LIN {X 0,Y 240.149,Z 451.003,A -85,B 0,C 180,E1 -19257.476,E2 -19257.476} C_VEL
LIN {X 0,Y 239.954,Z 446.945,A -85,B 0,C 180,E1 -19259.992,E2 -19259.992} C_VEL
LIN {X 0,Y 240.104,Z 441.489,A -85,B 0,C 180,E1 -19262.508,E2 -19262.508} C_VEL
LIN {X 0,Y 240.286,Z 435.643,A -85,B 0,C 180,E1 -19264.605,E2 -19264.605} C_VEL
LIN {X 0,Y 240.604,Z 428.331,A -85,B 0,C 180,E1 -19266.701,E2 -19266.701} C_VEL
LIN {X 0,Y 241.012,Z 420.068,A -85,B 0,C 180,E1 -19268.586,E2 -19268.586} C_VEL
LIN {X 0,Y 241.365,Z 412.286,A -85,B 0,C 180,E1 -19270.052,E2 -19270.052} C_VEL
LIN {X 0,Y 241.925,Z 402.905,A -85,B 0,C 180,E1 -19271.511,E2 -19271.511} C_VEL
LIN {X 0,Y 242.401,Z 391.7,A -85,B 0,C 180,E1 -19272.869,E2 -19272.869} C_VEL
LIN {X 0,Y 242.862,Z 381.433,A -85,B 0,C 180,E1 -19273.803,E2 -19273.803} C_VEL
LIN {X 0,Y 243.195,Z 370.502,A -85,B 0,C 180,E1 -19274.531,E2 -19274.531} C_VEL
LIN {X 0,Y 244.391,Z 317.786,A -85,B 0,C 180,E1 -19277.15,E2 -19277.15} C_VEL
LIN {X 0,Y 242.185,Z 296.983,A -85,B 0,C 180,E1 -19278.196,E2 -19278.196} C_VEL
LIN {X 0,Y 242.071,Z 295.173,A -85,B 0,C 180,E1 -19278.328,E2 -19278.328} C_VEL
LIN {X 0,Y 242.031,Z 295.147,A -85,B 0,C 180,E1 -19281.683,E2 -19281.683} C_VEL
LIN {X 0,Y 241.976,Z 295.155,A -85,B 0,C 180,E1 -19285.817,E2 -19285.817} C_VEL
LIN {X 0,Y 241.949,Z 295.156,A -85,B 0,C 180,E1 -19289.58,E2 -19289.58} C_VEL
LIN {X 0,Y 241.961,Z 295.154,A -85,B 0,C 180,E1 -19293.483,E2 -19293.483} C_VEL
LIN {X 0,Y 241.944,Z 295.157,A -85,B 0,C 180,E1 -19297.577,E2 -19297.577} C_VEL
LIN {X 0,Y 241.881,Z 295.164,A -85,B 0,C 180,E1 -19301.92,E2 -19301.92} C_VEL
LIN {X 0,Y 241.894,Z 295.166,A -85,B 0,C 180,E1 -19306.566,E2 -19306.566} C_VEL
LIN {X 0,Y 241.964,Z 295.155,A -85,B 0,C 180,E1 -19311.632,E2 -19311.632} C_VEL
LIN {X 0,Y 241.947,Z 295.158,A -85,B 0,C 180,E1 -19314.48,E2 -19314.48} C_VEL
LIN {X 0,Y 241.918,Z 295.158,A -85,B 0,C 180,E1 -19318.469,E2 -19318.469} C_VEL
LIN {X 0,Y 241.952,Z 295.156,A -85,B 0,C 180,E1 -19322.303,E2 -19322.303} C_VEL
LIN {X 0,Y 242,Z 295.149,A -85,B 0,C 180,E1 -19326.007,E2 -19326.007} C_VEL
LIN {X 0,Y 241.992,Z 295.154,A -85,B 0,C 180,E1 -19329.601,E2 -19329.601} C_VEL
LIN {X 0,Y 242.112,Z 295.139,A -85,B 0,C 180,E1 -19333.279,E2 -19333.279} C_VEL
LIN {X 0,Y 242.138,Z 295.133,A -85,B 0,C 180,E1 -19338.275,E2 -19338.275} C_VEL
LIN {X 0,Y 242.367,Z 295.109,A -85,B 0,C 180,E1 -19341.661,E2 -19341.661} C_VEL
LIN {X 0,Y 242.217,Z 295.121,A -85,B 0,C 180,E1 -19345.004,E2 -19345.004} C_VEL
LIN {X 0,Y 242.596,Z 295.078,A -85,B 0,C 180,E1 -19348.337,E2 -19348.337} C_VEL
LIN {X 0,Y 242.595,Z 295.078,A -85,B 0,C 180,E1 -19351.657,E2 -19351.657} C_VEL
LIN {X 0,Y 242.378,Z 295.104,A -85,B 0,C 180,E1 -19356.657,E2 -19356.657} C_VEL
LIN {X 0,Y 242.263,Z 295.12,A -85,B 0,C 180,E1 -19360.021,E2 -19360.021} C_VEL
LIN {X 0,Y 242.091,Z 295.138,A -85,B 0,C 180,E1 -19365.142,E2 -19365.142} C_VEL
LIN {X 0,Y 242.017,Z 295.152,A -85,B 0,C 180,E1 -19368.625,E2 -19368.625} C_VEL
LIN {X 0,Y 241.956,Z 295.155,A -85,B 0,C 180,E1 -19372.182,E2 -19372.182} C_VEL
LIN {X 0,Y 242.019,Z 295.148,A -85,B 0,C 180,E1 -19375.84,E2 -19375.84} C_VEL
LIN {X 0,Y 241.982,Z 295.152,A -85,B 0,C 180,E1 -19379.583,E2 -19379.583} C_VEL
LIN {X 0,Y 241.944,Z 295.158,A -85,B 0,C 180,E1 -19383.494,E2 -19383.494} C_VEL
LIN {X 0,Y 241.967,Z 295.155,A -85,B 0,C 180,E1 -19387.582,E2 -19387.582} C_VEL
LIN {X 0,Y 241.993,Z 295.15,A -85,B 0,C 180,E1 -19391.906,E2 -19391.906} C_VEL
LIN {X 0,Y 241.983,Z 295.153,A -85,B 0,C 180,E1 -19396.554,E2 -19396.554} C_VEL
LIN {X 0,Y 241.971,Z 295.152,A -85,B 0,C 180,E1 -19400.297,E2 -19400.297} C_VEL
LIN {X 0,Y 242,Z 295.15,A -85,B 0,C 180,E1 -19404.504,E2 -19404.504} C_VEL
LIN {X 0,Y 241.939,Z 295.155,A -85,B 0,C 180,E1 -19408.486,E2 -19408.486} C_VEL
LIN {X 0,Y 241.968,Z 295.155,A -85,B 0,C 180,E1 -19412.319,E2 -19412.319} C_VEL
LIN {X 0,Y 242.01,Z 295.15,A -85,B 0,C 180,E1 -19416.022,E2 -19416.022} C_VEL
LIN {X 0,Y 241.99,Z 295.152,A -85,B 0,C 180,E1 -19419.614,E2 -19419.614} C_VEL
LIN {X 0,Y 242.09,Z 295.139,A -85,B 0,C 180,E1 -19423.324,E2 -19423.324} C_VEL
LIN {X 0,Y 242.144,Z 295.136,A -85,B 0,C 180,E1 -19428.287,E2 -19428.287} C_VEL
LIN {X 0,Y 242.369,Z 295.105,A -85,B 0,C 180,E1 -19431.672,E2 -19431.672} C_VEL
LIN {X 0,Y 242.389,Z 295.101,A -85,B 0,C 180,E1 -19433.349,E2 -19433.349} C_VEL
LIN {X 0,Y 242.606,Z 295.078,A -85,B 0,C 180,E1 -19438.348,E2 -19438.348} C_VEL
LIN {X 0,Y 242.607,Z 295.074,A -85,B 0,C 180,E1 -19441.668,E2 -19441.668} C_VEL
LIN {X 0,Y 242.386,Z 295.105,A -85,B 0,C 180,E1 -19446.668,E2 -19446.668} C_VEL
LIN {X 0,Y 242.252,Z 295.119,A -85,B 0,C 180,E1 -19450.032,E2 -19450.032} C_VEL
LIN {X 0,Y 242.1,Z 295.14,A -85,B 0,C 180,E1 -19455.153,E2 -19455.153} C_VEL
LIN {X 0,Y 242.012,Z 295.151,A -85,B 0,C 180,E1 -19458.637,E2 -19458.637} C_VEL
LIN {X 0,Y 241.969,Z 295.151,A -85,B 0,C 180,E1 -19462.192,E2 -19462.192} C_VEL
LIN {X 0,Y 241.986,Z 295.153,A -85,B 0,C 180,E1 -19465.834,E2 -19465.834} C_VEL
LIN {X 0,Y 241.968,Z 295.155,A -85,B 0,C 180,E1 -19469.596,E2 -19469.596} C_VEL
LIN {X 0,Y 241.981,Z 295.156,A -85,B 0,C 180,E1 -19473.5,E2 -19473.5} C_VEL
LIN {X 0,Y 241.987,Z 295.155,A -85,B 0,C 180,E1 -19477.59,E2 -19477.59} C_VEL
LIN {X 0,Y 241.913,Z 295.163,A -85,B 0,C 180,E1 -19481.936,E2 -19481.936} C_VEL
LIN {X 0,Y 241.907,Z 295.162,A -85,B 0,C 180,E1 -19486.587,E2 -19486.587} C_VEL
LIN {X 0,Y 241.897,Z 295.161,A -85,B 0,C 180,E1 -19487.692,E2 -19487.692} C_VEL
LIN {X 0,Y 241.263,Z 295.244,A -85,B 0,C 180,E1 -19489.081,E2 -19489.081} C_VEL
LIN {X 0,Y 238.417,Z 295.599,A -85,B 0,C 180,E1 -19491.346,E2 -19491.346} C_VEL
LIN {X 0,Y 235.998,Z 295.898,A -85,B 0,C 180,E1 -19493.192,E2 -19493.192} C_VEL
LIN {X 0,Y 234.988,Z 296.025,A -85,B 0,C 180,E1 -19494.624,E2 -19494.624} C_VEL
LIN {X 0,Y 234.921,Z 296.032,A -85,B 0,C 180,E1 -19495.11,E2 -19495.11} C_VEL
LIN {X 0,Y 234.963,Z 296.026,A -85,B 0,C 180,E1 -19497.429,E2 -19497.429} C_VEL
LIN {X 0,Y 235.16,Z 296.003,A -85,B 0,C 180,E1 -19503.37,E2 -19503.37} C_VEL
LIN {X 0,Y 235.308,Z 296.003,A -85,B 0,C 180,E1 -19504.308,E2 -19504.308} C_VEL
LIN {X 0,Y 236.144,Z 300.672,A -85,B 0,C 180,E1 -19506.314,E2 -19506.314} C_VEL
LIN {X 0,Y 234.967,Z 310.218,A -85,B 0,C 180,E1 -19510.34,E2 -19510.34} C_VEL
LIN {X 0,Y 234.625,Z 313.396,A -85,B 0,C 180,E1 -19511.615,E2 -19511.615} C_VEL
LIN {X 0,Y 235.28,Z 331.783,A -85,B 0,C 180,E1 -19512.567,E2 -19512.567} C_VEL
LIN {X 0,Y 237.011,Z 351.619,A -85,B 0,C 180,E1 -19513.586,E2 -19513.586} C_VEL
LIN {X 0,Y 236.067,Z 391.667,A -85,B 0,C 180,E1 -19515.73,E2 -19515.73} C_VEL
LIN {X 0,Y 235.686,Z 404.414,A -85,B 0,C 180,E1 -19516.751,E2 -19516.751} C_VEL
LIN {X 0,Y 235.205,Z 414.901,A -85,B 0,C 180,E1 -19517.93,E2 -19517.93} C_VEL
LIN {X 0,Y 234.653,Z 425.377,A -85,B 0,C 180,E1 -19519.432,E2 -19519.432} C_VEL
LIN {X 0,Y 234.32,Z 434.778,A -85,B 0,C 180,E1 -19521.161,E2 -19521.161} C_VEL
LIN {X 0,Y 234.06,Z 442.15,A -85,B 0,C 180,E1 -19522.833,E2 -19522.833} C_VEL
LIN {X 0,Y 233.943,Z 447.951,A -85,B 0,C 180,E1 -19524.4,E2 -19524.4} C_VEL
LIN {X 0,Y 233.806,Z 453.277,A -85,B 0,C 180,E1 -19526.125,E2 -19526.125} C_VEL
LIN {X 0,Y 233.634,Z 458.627,A -85,B 0,C 180,E1 -19528.279,E2 -19528.279} C_VEL
LIN {X 0,Y 233.647,Z 462.032,A -85,B 0,C 180,E1 -19530.003,E2 -19530.003} C_VEL
LIN {X 0,Y 233.127,Z 465.79,A -85,B 0,C 180,E1 -19532.595,E2 -19532.595} C_VEL
LIN {X 0,Y 233.083,Z 466.846,A -85,B 0,C 180,E1 -19533.46,E2 -19533.46} C_VEL
LIN {X 0,Y 233.017,Z 468.599,A -85,B 0,C 180,E1 -19535.496,E2 -19535.496} C_VEL
LIN {X 0,Y 233.483,Z 469.925,A -85,B 0,C 180,E1 -19538.659,E2 -19538.659} C_VEL
LIN {X 0,Y 234.1,Z 470.04,A -85,B 0,C 180,E1 -19540.38,E2 -19540.38} C_VEL
LIN {X 0,Y 235.015,Z 469.572,A -85,B 0,C 180,E1 -19542.086,E2 -19542.086} C_VEL
LIN {X 0,Y 236.181,Z 468.648,A -85,B 0,C 180,E1 -19543.775,E2 -19543.775} C_VEL
LIN {X 0,Y 237.612,Z 467.294,A -85,B 0,C 180,E1 -19545.441,E2 -19545.441} C_VEL
LIN {X 0,Y 240.273,Z 464.246,A -85,B 0,C 180,E1 -19547.889,E2 -19547.889} C_VEL
LIN {X 0,Y 243.332,Z 459.986,A -85,B 0,C 180,E1 -19550.281,E2 -19550.281} C_VEL
LIN {X 0,Y 247.114,Z 454.428,A -85,B 0,C 180,E1 -19552.581,E2 -19552.581} C_VEL
LIN {X 0,Y 251.451,Z 447.192,A -85,B 0,C 180,E1 -19554.79,E2 -19554.79} C_VEL
LIN {X 0,Y 255.482,Z 439.593,A -85,B 0,C 180,E1 -19556.555,E2 -19556.555} C_VEL
LIN {X 0,Y 259.012,Z 432.389,A -85,B 0,C 180,E1 -19557.911,E2 -19557.911} C_VEL
LIN {X 0,Y 263.323,Z 422.543,A -85,B 0,C 180,E1 -19559.371,E2 -19559.371} C_VEL
LIN {X 0,Y 266.874,Z 412.869,A -85,B 0,C 180,E1 -19560.463,E2 -19560.463} C_VEL
LIN {X 0,Y 270.66,Z 400.767,A -85,B 0,C 180,E1 -19561.507,E2 -19561.507} C_VEL
LIN {X 0,Y 273.795,Z 387.59,A -85,B 0,C 180,E1 -19562.349,E2 -19562.349} C_VEL
LIN {X 0,Y 277.03,Z 368.395,A -85,B 0,C 180,E1 -19563.328,E2 -19563.328} C_VEL
LIN {X 0,Y 276.992,Z 361.037,A -85,B 0,C 180,E1 -19564.254,E2 -19564.254} C_VEL
LIN {X 0,Y 275.534,Z 356.361,A -85,B 0,C 180,E1 -19565.635,E2 -19565.635} C_VEL
LIN {X 0,Y 274.342,Z 352.867,A -85,B 0,C 180,E1 -19566.887,E2 -19566.887} C_VEL
LIN {X 0,Y 272.769,Z 348.624,A -85,B 0,C 180,E1 -19568.806,E2 -19568.806} C_VEL
LIN {X 0,Y 271.252,Z 344.781,A -85,B 0,C 180,E1 -19571.46,E2 -19571.46} C_VEL
LIN {X 0,Y 270.741,Z 343.145,A -85,B 0,C 180,E1 -19573.004,E2 -19573.004} C_VEL
LIN {X 0,Y 270.453,Z 342.213,A -85,B 0,C 180,E1 -19575.435,E2 -19575.435} C_VEL
LIN {X 0,Y 270.947,Z 342.366,A -85,B 0,C 180,E1 -19577.894,E2 -19577.894} C_VEL
LIN {X 0,Y 272.784,Z 344.473,A -85,B 0,C 180,E1 -19581.133,E2 -19581.133} C_VEL
LIN {X 0,Y 275.194,Z 348.814,A -85,B 0,C 180,E1 -19583.901,E2 -19583.901} C_VEL
LIN {X 0,Y 277.423,Z 353.09,A -85,B 0,C 180,E1 -19585.804,E2 -19585.804} C_VEL
LIN {X 0,Y 278.716,Z 356.282,A -85,B 0,C 180,E1 -19586.86,E2 -19586.86} C_VEL
LIN {X 0,Y 274.25,Z 381.604,A -85,B 0,C 180,E1 -19588.122,E2 -19588.122} C_VEL
LIN {X 0,Y 271.351,Z 393.478,A -85,B 0,C 180,E1 -19588.99,E2 -19588.99} C_VEL
LIN {X 0,Y 268.372,Z 403.254,A -85,B 0,C 180,E1 -19589.938,E2 -19589.938} C_VEL
LIN {X 0,Y 264.75,Z 413.627,A -85,B 0,C 180,E1 -19591.233,E2 -19591.233} C_VEL
LIN {X 0,Y 260.819,Z 422.792,A -85,B 0,C 180,E1 -19592.73,E2 -19592.73} C_VEL
LIN {X 0,Y 257.513,Z 429.527,A -85,B 0,C 180,E1 -19594.101,E2 -19594.101} C_VEL
LIN {X 0,Y 253.687,Z 436.569,A -85,B 0,C 180,E1 -19595.874,E2 -19595.874} C_VEL
LIN {X 0,Y 250.208,Z 442.258,A -85,B 0,C 180,E1 -19597.709,E2 -19597.709} C_VEL
LIN {X 0,Y 246.361,Z 447.517,A -85,B 0,C 180,E1 -19599.974,E2 -19599.974} C_VEL
LIN {X 0,Y 242.974,Z 451.443,A -85,B 0,C 180,E1 -19602.312,E2 -19602.312} C_VEL
LIN {X 0,Y 240.013,Z 454.144,A -85,B 0,C 180,E1 -19604.712,E2 -19604.712} C_VEL
LIN {X 0,Y 238.332,Z 455.272,A -85,B 0,C 180,E1 -19606.347,E2 -19606.347} C_VEL
LIN {X 0,Y 237.062,Z 455.939,A -85,B 0,C 180,E1 -19608.015,E2 -19608.015} C_VEL
LIN {X 0,Y 235.74,Z 456.104,A -85,B 0,C 180,E1 -19609.688,E2 -19609.688} C_VEL
LIN {X 0,Y 234.712,Z 455.683,A -85,B 0,C 180,E1 -19611.381,E2 -19611.381} C_VEL
LIN {X 0,Y 234.014,Z 454.806,A -85,B 0,C 180,E1 -19613.092,E2 -19613.092} C_VEL
LIN {X 0,Y 233.564,Z 453.485,A -85,B 0,C 180,E1 -19614.812,E2 -19614.812} C_VEL
LIN {X 0,Y 233.249,Z 451.636,A -85,B 0,C 180,E1 -19616.537,E2 -19616.537} C_VEL
LIN {X 0,Y 232.909,Z 447.69,A -85,B 0,C 180,E1 -19619.127,E2 -19619.127} C_VEL
LIN {X 0,Y 232.987,Z 442.366,A -85,B 0,C 180,E1 -19621.72,E2 -19621.72} C_VEL
LIN {X 0,Y 233.23,Z 436.729,A -85,B 0,C 180,E1 -19623.879,E2 -19623.879} C_VEL
LIN {X 0,Y 233.48,Z 429.049,A -85,B 0,C 180,E1 -19626.217,E2 -19626.217} C_VEL
LIN {X 0,Y 233.906,Z 420.7,A -85,B 0,C 180,E1 -19628.196,E2 -19628.196} C_VEL
LIN {X 0,Y 234.329,Z 411.768,A -85,B 0,C 180,E1 -19629.921,E2 -19629.921} C_VEL
LIN {X 0,Y 234.95,Z 400.646,A -85,B 0,C 180,E1 -19631.639,E2 -19631.639} C_VEL
LIN {X 0,Y 235.424,Z 389.561,A -85,B 0,C 180,E1 -19632.928,E2 -19632.928} C_VEL
LIN {X 0,Y 235.899,Z 378.809,A -85,B 0,C 180,E1 -19633.889,E2 -19633.889} C_VEL
LIN {X 0,Y 236.287,Z 362.692,A -85,B 0,C 180,E1 -19634.855,E2 -19634.855} C_VEL
LIN {X 0,Y 237.251,Z 318.134,A -85,B 0,C 180,E1 -19637.166,E2 -19637.166} C_VEL
LIN {X 0,Y 235.101,Z 296.963,A -85,B 0,C 180,E1 -19638.257,E2 -19638.257} C_VEL
LIN {X 0,Y 235.028,Z 296.023,A -85,B 0,C 180,E1 -19638.35,E2 -19638.35} C_VEL
LIN {X 0,Y 234.987,Z 296.025,A -85,B 0,C 180,E1 -19642,E2 -19642} C_VEL
LIN {X 0,Y 234.911,Z 296.035,A -85,B 0,C 180,E1 -19646.653,E2 -19646.653} C_VEL
LIN {X 0,Y 234.88,Z 296.037,A -85,B 0,C 180,E1 -19650.563,E2 -19650.563} C_VEL
LIN {X 0,Y 234.904,Z 296.038,A -85,B 0,C 180,E1 -19654.63,E2 -19654.63} C_VEL
LIN {X 0,Y 234.891,Z 296.036,A -85,B 0,C 180,E1 -19658.925,E2 -19658.925} C_VEL
LIN {X 0,Y 234.843,Z 296.042,A -85,B 0,C 180,E1 -19664.088,E2 -19664.088} C_VEL
LIN {X 0,Y 234.843,Z 296.042,A -85,B 0,C 180,E1 -19668.414,E2 -19668.414} C_VEL
LIN {X 0,Y 234.888,Z 296.039,A -85,B 0,C 180,E1 -19671.07,E2 -19671.07} C_VEL
LIN {X 0,Y 234.893,Z 296.037,A -85,B 0,C 180,E1 -19675.353,E2 -19675.353} C_VEL
LIN {X 0,Y 234.866,Z 296.04,A -85,B 0,C 180,E1 -19679.42,E2 -19679.42} C_VEL
LIN {X 0,Y 234.955,Z 296.029,A -85,B 0,C 180,E1 -19683.787,E2 -19683.787} C_VEL
LIN {X 0,Y 234.956,Z 296.027,A -85,B 0,C 180,E1 -19688.962,E2 -19688.962} C_VEL
LIN {X 0,Y 235.047,Z 296.018,A -85,B 0,C 180,E1 -19693.06,E2 -19693.06} C_VEL
LIN {X 0,Y 235.069,Z 296.015,A -85,B 0,C 180,E1 -19697.917,E2 -19697.917} C_VEL
LIN {X 0,Y 235.299,Z 295.987,A -85,B 0,C 180,E1 -19701.408,E2 -19701.408} C_VEL
LIN {X 0,Y 235.332,Z 295.981,A -85,B 0,C 180,E1 -19703.136,E2 -19703.136} C_VEL
LIN {X 0,Y 235.557,Z 295.955,A -85,B 0,C 180,E1 -19708.287,E2 -19708.287} C_VEL
LIN {X 0,Y 235.556,Z 295.955,A -85,B 0,C 180,E1 -19711.707,E2 -19711.707} C_VEL
LIN {X 0,Y 235.329,Z 295.981,A -85,B 0,C 180,E1 -19716.858,E2 -19716.858} C_VEL
LIN {X 0,Y 235.187,Z 296.003,A -85,B 0,C 180,E1 -19720.326,E2 -19720.326} C_VEL
LIN {X 0,Y 235.045,Z 296.016,A -85,B 0,C 180,E1 -19725.608,E2 -19725.608} C_VEL
LIN {X 0,Y 234.954,Z 296.028,A -85,B 0,C 180,E1 -19729.207,E2 -19729.207} C_VEL
LIN {X 0,Y 234.903,Z 296.035,A -85,B 0,C 180,E1 -19732.885,E2 -19732.885} C_VEL
LIN {X 0,Y 234.921,Z 296.036,A -85,B 0,C 180,E1 -19736.66,E2 -19736.66} C_VEL
LIN {X 0,Y 234.884,Z 296.038,A -85,B 0,C 180,E1 -19740.571,E2 -19740.571} C_VEL
LIN {X 0,Y 234.915,Z 296.034,A -85,B 0,C 180,E1 -19744.637,E2 -19744.637} C_VEL
LIN {X 0,Y 234.923,Z 296.035,A -85,B 0,C 180,E1 -19748.956,E2 -19748.956} C_VEL
LIN {X 0,Y 234.953,Z 296.031,A -85,B 0,C 180,E1 -19753.466,E2 -19753.466} C_VEL
LIN {X 0,Y 234.955,Z 296.028,A -85,B 0,C 180,E1 -19756.545,E2 -19756.545} C_VEL
LIN {X 0,Y 234.917,Z 296.033,A -85,B 0,C 180,E1 -19761.092,E2 -19761.092} C_VEL
LIN {X 0,Y 234.924,Z 296.035,A -85,B 0,C 180,E1 -19765.374,E2 -19765.374} C_VEL
LIN {X 0,Y 234.888,Z 296.036,A -85,B 0,C 180,E1 -19769.438,E2 -19769.438} C_VEL
LIN {X 0,Y 234.962,Z 296.031,A -85,B 0,C 180,E1 -19773.802,E2 -19773.802} C_VEL
LIN {X 0,Y 234.941,Z 296.028,A -85,B 0,C 180,E1 -19778.974,E2 -19778.974} C_VEL
LIN {X 0,Y 235.031,Z 296.018,A -85,B 0,C 180,E1 -19783.1,E2 -19783.1} C_VEL
LIN {X 0,Y 235.076,Z 296.013,A -85,B 0,C 180,E1 -19787.93,E2 -19787.93} C_VEL
LIN {X 0,Y 235.302,Z 295.985,A -85,B 0,C 180,E1 -19791.421,E2 -19791.421} C_VEL
LIN {X 0,Y 235.341,Z 295.979,A -85,B 0,C 180,E1 -19793.149,E2 -19793.149} C_VEL
LIN {X 0,Y 235.564,Z 295.954,A -85,B 0,C 180,E1 -19798.299,E2 -19798.299} C_VEL
LIN {X 0,Y 235.566,Z 295.952,A -85,B 0,C 180,E1 -19801.718,E2 -19801.718} C_VEL
LIN {X 0,Y 235.337,Z 295.983,A -85,B 0,C 180,E1 -19806.869,E2 -19806.869} C_VEL
LIN {X 0,Y 235.199,Z 295.999,A -85,B 0,C 180,E1 -19810.336,E2 -19810.336} C_VEL
LIN {X 0,Y 235.036,Z 296.018,A -85,B 0,C 180,E1 -19815.62,E2 -19815.62} C_VEL
LIN {X 0,Y 234.954,Z 296.031,A -85,B 0,C 180,E1 -19819.218,E2 -19819.218} C_VEL
LIN {X 0,Y 234.906,Z 296.034,A -85,B 0,C 180,E1 -19822.896,E2 -19822.896} C_VEL
LIN {X 0,Y 234.924,Z 296.033,A -85,B 0,C 180,E1 -19826.671,E2 -19826.671} C_VEL
LIN {X 0,Y 234.899,Z 296.033,A -85,B 0,C 180,E1 -19830.58,E2 -19830.58} C_VEL
LIN {X 0,Y 234.925,Z 296.031,A -85,B 0,C 180,E1 -19834.647,E2 -19834.647} C_VEL
LIN {X 0,Y 234.917,Z 296.032,A -85,B 0,C 180,E1 -19838.942,E2 -19838.942} C_VEL
LIN {X 0,Y 234.859,Z 296.042,A -85,B 0,C 180,E1 -19843.501,E2 -19843.501} C_VEL
LIN {X 0,Y 234.829,Z 296.039,A -85,B 0,C 180,E1 -19847.699,E2 -19847.699} C_VEL
LIN {X 0,Y 234.928,Z 296.03,A -85,B 0,C 180,E1 -19851.085,E2 -19851.085} C_VEL
LIN {X 0,Y 234.921,Z 296.032,A -85,B 0,C 180,E1 -19855.11,E2 -19855.11} C_VEL
LIN {X 0,Y 234.284,Z 296.115,A -85,B 0,C 180,E1 -19856.541,E2 -19856.541} C_VEL
LIN {X 0,Y 231.42,Z 296.477,A -85,B 0,C 180,E1 -19858.877,E2 -19858.877} C_VEL
LIN {X 0,Y 229.019,Z 296.775,A -85,B 0,C 180,E1 -19860.782,E2 -19860.782} C_VEL
LIN {X 0,Y 228.068,Z 296.89,A -85,B 0,C 180,E1 -19862.261,E2 -19862.261} C_VEL
LIN {X 0,Y 228.033,Z 296.891,A -85,B 0,C 180,E1 -19862.761,E2 -19862.761} C_VEL
LIN {X 0,Y 228.329,Z 297.049,A -85,B 0,C 180,E1 -19864.6,E2 -19864.6} C_VEL
LIN {X 0,Y 229.014,Z 301.34,A -85,B 0,C 180,E1 -19866.491,E2 -19866.491} C_VEL
LIN {X 0,Y 227.653,Z 311.864,A -85,B 0,C 180,E1 -19871.089,E2 -19871.089} C_VEL
LIN {X 0,Y 227.549,Z 312.905,A -85,B 0,C 180,E1 -19871.547,E2 -19871.547} C_VEL
LIN {X 0,Y 228.135,Z 331.437,A -85,B 0,C 180,E1 -19872.566,E2 -19872.566} C_VEL
LIN {X 0,Y 229.906,Z 351.989,A -85,B 0,C 180,E1 -19873.671,E2 -19873.671} C_VEL
LIN {X 0,Y 228.989,Z 392.539,A -85,B 0,C 180,E1 -19875.96,E2 -19875.96} C_VEL
LIN {X 0,Y 228.634,Z 404.811,A -85,B 0,C 180,E1 -19877.013,E2 -19877.013} C_VEL
LIN {X 0,Y 228.132,Z 415.129,A -85,B 0,C 180,E1 -19878.227,E2 -19878.227} C_VEL
LIN {X 0,Y 227.596,Z 425.497,A -85,B 0,C 180,E1 -19879.776,E2 -19879.776} C_VEL
LIN {X 0,Y 227.31,Z 435.35,A -85,B 0,C 180,E1 -19881.681,E2 -19881.681} C_VEL
LIN {X 0,Y 227.086,Z 442.336,A -85,B 0,C 180,E1 -19883.339,E2 -19883.339} C_VEL
LIN {X 0,Y 226.939,Z 448.507,A -85,B 0,C 180,E1 -19885.118,E2 -19885.118} C_VEL
LIN {X 0,Y 226.793,Z 453.602,A -85,B 0,C 180,E1 -19886.894,E2 -19886.894} C_VEL
LIN {X 0,Y 226.711,Z 458.772,A -85,B 0,C 180,E1 -19889.115,E2 -19889.115} C_VEL
LIN {X 0,Y 226.48,Z 462.012,A -85,B 0,C 180,E1 -19890.892,E2 -19890.892} C_VEL
LIN {X 0,Y 226.094,Z 465.69,A -85,B 0,C 180,E1 -19893.567,E2 -19893.567} C_VEL
LIN {X 0,Y 226.023,Z 467.642,A -85,B 0,C 180,E1 -19895.667,E2 -19895.667} C_VEL
LIN {X 0,Y 226.129,Z 468.648,A -85,B 0,C 180,E1 -19897.144,E2 -19897.144} C_VEL
LIN {X 0,Y 226.48,Z 469.419,A -85,B 0,C 180,E1 -19898.929,E2 -19898.929} C_VEL
LIN {X 0,Y 227.126,Z 469.628,A -85,B 0,C 180,E1 -19900.702,E2 -19900.702} C_VEL
LIN {X 0,Y 228.076,Z 469.411,A -85,B 0,C 180,E1 -19902.459,E2 -19902.459} C_VEL
LIN {X 0,Y 229.289,Z 468.783,A -85,B 0,C 180,E1 -19904.197,E2 -19904.197} C_VEL
LIN {X 0,Y 230.807,Z 467.623,A -85,B 0,C 180,E1 -19905.908,E2 -19905.908} C_VEL
LIN {X 0,Y 233.558,Z 464.956,A -85,B 0,C 180,E1 -19908.421,E2 -19908.421} C_VEL
LIN {X 0,Y 236.777,Z 461.113,A -85,B 0,C 180,E1 -19910.869,E2 -19910.869} C_VEL
LIN {X 0,Y 239.315,Z 457.882,A -85,B 0,C 180,E1 -19912.446,E2 -19912.446} C_VEL
LIN {X 0,Y 243.636,Z 451.654,A -85,B 0,C 180,E1 -19914.728,E2 -19914.728} C_VEL
LIN {X 0,Y 247.68,Z 445.304,A -85,B 0,C 180,E1 -19916.548,E2 -19916.548} C_VEL
LIN {X 0,Y 252.05,Z 437.548,A -85,B 0,C 180,E1 -19918.298,E2 -19918.298} C_VEL
LIN {X 0,Y 256.869,Z 427.868,A -85,B 0,C 180,E1 -19919.958,E2 -19919.958} C_VEL
LIN {X 0,Y 261.048,Z 418.282,A -85,B 0,C 180,E1 -19921.218,E2 -19921.218} C_VEL
LIN {X 0,Y 264.939,Z 407.932,A -85,B 0,C 180,E1 -19922.269,E2 -19922.269} C_VEL
LIN {X 0,Y 268.66,Z 395.432,A -85,B 0,C 180,E1 -19923.213,E2 -19923.213} C_VEL
LIN {X 0,Y 271.641,Z 382.131,A -85,B 0,C 180,E1 -19923.973,E2 -19923.973} C_VEL
LIN {X 0,Y 273.685,Z 370.456,A -85,B 0,C 180,E1 -19924.572,E2 -19924.572} C_VEL
LIN {X 0,Y 273.736,Z 365.472,A -85,B 0,C 180,E1 -19925.245,E2 -19925.245} C_VEL
LIN {X 0,Y 272.489,Z 361.188,A -85,B 0,C 180,E1 -19926.597,E2 -19926.597} C_VEL
LIN {X 0,Y 270.977,Z 356.51,A -85,B 0,C 180,E1 -19928.498,E2 -19928.498} C_VEL
LIN {X 0,Y 269.845,Z 353.298,A -85,B 0,C 180,E1 -19930.356,E2 -19930.356} C_VEL
LIN {X 0,Y 268.955,Z 350.255,A -85,B 0,C 180,E1 -19932.799,E2 -19932.799} C_VEL
LIN {X 0,Y 268.65,Z 349.106,A -85,B 0,C 180,E1 -19935.055,E2 -19935.055} C_VEL
LIN {X 0,Y 269.134,Z 349.278,A -85,B 0,C 180,E1 -19937.959,E2 -19937.959} C_VEL
LIN {X 0,Y 270.799,Z 351.271,A -85,B 0,C 180,E1 -19940.991,E2 -19940.991} C_VEL
LIN {X 0,Y 272.856,Z 355.347,A -85,B 0,C 180,E1 -19943.542,E2 -19943.542} C_VEL
LIN {X 0,Y 274.645,Z 359.009,A -85,B 0,C 180,E1 -19945.221,E2 -19945.221} C_VEL
LIN {X 0,Y 275.179,Z 360.272,A -85,B 0,C 180,E1 -19945.681,E2 -19945.681} C_VEL
LIN {X 0,Y 270.908,Z 382.52,A -85,B 0,C 180,E1 -19946.821,E2 -19946.821} C_VEL
LIN {X 0,Y 267.877,Z 394.097,A -85,B 0,C 180,E1 -19947.668,E2 -19947.668} C_VEL
LIN {X 0,Y 264.796,Z 403.788,A -85,B 0,C 180,E1 -19948.602,E2 -19948.602} C_VEL
LIN {X 0,Y 260.928,Z 413.997,A -85,B 0,C 180,E1 -19949.883,E2 -19949.883} C_VEL
LIN {X 0,Y 256.734,Z 423.055,A -85,B 0,C 180,E1 -19951.369,E2 -19951.369} C_VEL
LIN {X 0,Y 253.228,Z 429.848,A -85,B 0,C 180,E1 -19952.739,E2 -19952.739} C_VEL
LIN {X 0,Y 249.282,Z 436.553,A -85,B 0,C 180,E1 -19954.428,E2 -19954.428} C_VEL
LIN {X 0,Y 245.327,Z 442.483,A -85,B 0,C 180,E1 -19956.348,E2 -19956.348} C_VEL
LIN {X 0,Y 241.214,Z 447.812,A -85,B 0,C 180,E1 -19958.634,E2 -19958.634} C_VEL
LIN {X 0,Y 237.48,Z 451.729,A -85,B 0,C 180,E1 -19960.994,E2 -19960.994} C_VEL
LIN {X 0,Y 235.284,Z 453.687,A -85,B 0,C 180,E1 -19962.612,E2 -19962.612} C_VEL
LIN {X 0,Y 233.25,Z 455.158,A -85,B 0,C 180,E1 -19964.258,E2 -19964.258} C_VEL
LIN {X 0,Y 231.484,Z 456.018,A -85,B 0,C 180,E1 -19965.935,E2 -19965.935} C_VEL
LIN {X 0,Y 230.146,Z 456.389,A -85,B 0,C 180,E1 -19967.649,E2 -19967.649} C_VEL
LIN {X 0,Y 228.207,Z 456.092,A -85,B 0,C 180,E1 -19970.241,E2 -19970.241} C_VEL
LIN {X 0,Y 226.976,Z 454.69,A -85,B 0,C 180,E1 -19972.877,E2 -19972.877} C_VEL
LIN {X 0,Y 226.338,Z 452.181,A -85,B 0,C 180,E1 -19975.539,E2 -19975.539} C_VEL
LIN {X 0,Y 225.918,Z 448.417,A -85,B 0,C 180,E1 -19978.208,E2 -19978.208} C_VEL
LIN {X 0,Y 225.886,Z 443.195,A -85,B 0,C 180,E1 -19980.882,E2 -19980.882} C_VEL
LIN {X 0,Y 226.161,Z 437.68,A -85,B 0,C 180,E1 -19983.108,E2 -19983.108} C_VEL
LIN {X 0,Y 226.322,Z 430.798,A -85,B 0,C 180,E1 -19985.336,E2 -19985.336} C_VEL
LIN {X 0,Y 226.773,Z 422.436,A -85,B 0,C 180,E1 -19987.514,E2 -19987.514} C_VEL
LIN {X 0,Y 227.204,Z 413.652,A -85,B 0,C 180,E1 -19989.336,E2 -19989.336} C_VEL
LIN {X 0,Y 227.593,Z 405.859,A -85,B 0,C 180,E1 -19990.668,E2 -19990.668} C_VEL
LIN {X 0,Y 228.039,Z 396.326,A -85,B 0,C 180,E1 -19991.997,E2 -19991.997} C_VEL
LIN {X 0,Y 228.65,Z 383.974,A -85,B 0,C 180,E1 -19993.318,E2 -19993.318} C_VEL
LIN {X 0,Y 228.977,Z 373.057,A -85,B 0,C 180,E1 -19994.147,E2 -19994.147} C_VEL
LIN {X 0,Y 230.251,Z 319.215,A -85,B 0,C 180,E1 -19997.103,E2 -19997.103} C_VEL
LIN {X 0,Y 228.045,Z 298.255,A -85,B 0,C 180,E1 -19998.23,E2 -19998.23} C_VEL
LIN {X 0,Y 227.997,Z 296.899,A -85,B 0,C 180,E1 -19998.35,E2 -19998.35} C_VEL
LIN {X 0,Y 227.912,Z 296.905,A -85,B 0,C 180,E1 -20002.312,E2 -20002.312} C_VEL
LIN {X 0,Y 227.89,Z 296.91,A -85,B 0,C 180,E1 -20006.571,E2 -20006.571} C_VEL
LIN {X 0,Y 227.855,Z 296.914,A -85,B 0,C 180,E1 -20010.268,E2 -20010.268} C_VEL
LIN {X 0,Y 227.859,Z 296.911,A -85,B 0,C 180,E1 -20013.711,E2 -20013.711} C_VEL
LIN {X 0,Y 227.817,Z 296.918,A -85,B 0,C 180,E1 -20018.083,E2 -20018.083} C_VEL
LIN {X 0,Y 227.761,Z 296.927,A -85,B 0,C 180,E1 -20022.739,E2 -20022.739} C_VEL
LIN {X 0,Y 227.773,Z 296.923,A -85,B 0,C 180,E1 -20027.246,E2 -20027.246} C_VEL
LIN {X 0,Y 227.81,Z 296.917,A -85,B 0,C 180,E1 -20031.899,E2 -20031.899} C_VEL
LIN {X 0,Y 227.845,Z 296.913,A -85,B 0,C 180,E1 -20036.369,E2 -20036.369} C_VEL
LIN {X 0,Y 227.847,Z 296.912,A -85,B 0,C 180,E1 -20040.425,E2 -20040.425} C_VEL
LIN {X 0,Y 227.886,Z 296.908,A -85,B 0,C 180,E1 -20044.418,E2 -20044.418} C_VEL
LIN {X 0,Y 227.907,Z 296.904,A -85,B 0,C 180,E1 -20048.279,E2 -20048.279} C_VEL
LIN {X 0,Y 227.987,Z 296.897,A -85,B 0,C 180,E1 -20052.825,E2 -20052.825} C_VEL
LIN {X 0,Y 228.025,Z 296.891,A -85,B 0,C 180,E1 -20057.538,E2 -20057.538} C_VEL
LIN {X 0,Y 228.235,Z 296.866,A -85,B 0,C 180,E1 -20061.14,E2 -20061.14} C_VEL
LIN {X 0,Y 228.284,Z 296.859,A -85,B 0,C 180,E1 -20062.923,E2 -20062.923} C_VEL
LIN {X 0,Y 228.516,Z 296.832,A -85,B 0,C 180,E1 -20068.235,E2 -20068.235} C_VEL
LIN {X 0,Y 228.515,Z 296.832,A -85,B 0,C 180,E1 -20071.759,E2 -20071.759} C_VEL
LIN {X 0,Y 228.28,Z 296.859,A -85,B 0,C 180,E1 -20077.071,E2 -20077.071} C_VEL
LIN {X 0,Y 228.109,Z 296.882,A -85,B 0,C 180,E1 -20080.65,E2 -20080.65} C_VEL
LIN {X 0,Y 227.995,Z 296.896,A -85,B 0,C 180,E1 -20086.103,E2 -20086.103} C_VEL
LIN {X 0,Y 227.885,Z 296.909,A -85,B 0,C 180,E1 -20089.827,E2 -20089.827} C_VEL
LIN {X 0,Y 227.857,Z 296.91,A -85,B 0,C 180,E1 -20093.635,E2 -20093.635} C_VEL
LIN {X 0,Y 227.837,Z 296.915,A -85,B 0,C 180,E1 -20097.558,E2 -20097.558} C_VEL
LIN {X 0,Y 227.826,Z 296.913,A -85,B 0,C 180,E1 -20101.625,E2 -20101.625} C_VEL
LIN {X 0,Y 227.856,Z 296.913,A -85,B 0,C 180,E1 -20105.872,E2 -20105.872} C_VEL
LIN {X 0,Y 227.86,Z 296.909,A -85,B 0,C 180,E1 -20110.365,E2 -20110.365} C_VEL
LIN {X 0,Y 227.878,Z 296.911,A -85,B 0,C 180,E1 -20114.834,E2 -20114.834} C_VEL
LIN {X 0,Y 227.886,Z 296.908,A -85,B 0,C 180,E1 -20117.74,E2 -20117.74} C_VEL
LIN {X 0,Y 227.833,Z 296.916,A -85,B 0,C 180,E1 -20121.921,E2 -20121.921} C_VEL
LIN {X 0,Y 227.854,Z 296.911,A -85,B 0,C 180,E1 -20126.38,E2 -20126.38} C_VEL
LIN {X 0,Y 227.871,Z 296.91,A -85,B 0,C 180,E1 -20130.443,E2 -20130.443} C_VEL
LIN {X 0,Y 227.894,Z 296.908,A -85,B 0,C 180,E1 -20134.433,E2 -20134.433} C_VEL
LIN {X 0,Y 227.91,Z 296.905,A -85,B 0,C 180,E1 -20138.293,E2 -20138.293} C_VEL
LIN {X 0,Y 227.999,Z 296.898,A -85,B 0,C 180,E1 -20143.904,E2 -20143.904} C_VEL
LIN {X 0,Y 228.034,Z 296.888,A -85,B 0,C 180,E1 -20147.551,E2 -20147.551} C_VEL
LIN {X 0,Y 228.24,Z 296.865,A -85,B 0,C 180,E1 -20151.153,E2 -20151.153} C_VEL
LIN {X 0,Y 228.292,Z 296.858,A -85,B 0,C 180,E1 -20152.936,E2 -20152.936} C_VEL
LIN {X 0,Y 228.523,Z 296.831,A -85,B 0,C 180,E1 -20158.247,E2 -20158.247} C_VEL
LIN {X 0,Y 228.525,Z 296.829,A -85,B 0,C 180,E1 -20161.771,E2 -20161.771} C_VEL
LIN {X 0,Y 228.289,Z 296.86,A -85,B 0,C 180,E1 -20167.082,E2 -20167.082} C_VEL
LIN {X 0,Y 228.13,Z 296.882,A -85,B 0,C 180,E1 -20170.66,E2 -20170.66} C_VEL
LIN {X 0,Y 227.994,Z 296.895,A -85,B 0,C 180,E1 -20176.115,E2 -20176.115} C_VEL
LIN {X 0,Y 227.915,Z 296.902,A -85,B 0,C 180,E1 -20181.726,E2 -20181.726} C_VEL
LIN {X 0,Y 227.902,Z 296.907,A -85,B 0,C 180,E1 -20186.59,E2 -20186.59} C_VEL
LIN {X 0,Y 227.874,Z 296.908,A -85,B 0,C 180,E1 -20190.288,E2 -20190.288} C_VEL
LIN {X 0,Y 227.879,Z 296.911,A -85,B 0,C 180,E1 -20193.729,E2 -20193.729} C_VEL
LIN {X 0,Y 227.845,Z 296.913,A -85,B 0,C 180,E1 -20198.1,E2 -20198.1} C_VEL
LIN {X 0,Y 227.791,Z 296.919,A -85,B 0,C 180,E1 -20202.756,E2 -20202.756} C_VEL
LIN {X 0,Y 227.793,Z 296.921,A -85,B 0,C 180,E1 -20207.258,E2 -20207.258} C_VEL
LIN {X 0,Y 227.85,Z 296.916,A -85,B 0,C 180,E1 -20211.915,E2 -20211.915} C_VEL
LIN {X 0,Y 227.89,Z 296.908,A -85,B 0,C 180,E1 -20216.384,E2 -20216.384} C_VEL
LIN {X 0,Y 227.902,Z 296.909,A -85,B 0,C 180,E1 -20220.439,E2 -20220.439} C_VEL
LIN {X 0,Y 228.033,Z 296.891,A -85,B 0,C 180,E1 -20222.761,E2 -20222.761} C_VEL
LIN {X 0,Y 227.814,Z 297.268,A -85,B 0,C 180,E1 -20223.739,E2 -20223.739} C_VEL
LIN {X 0,Y 227.098,Z 298.266,A -85,B 0,C 180,E1 -20224.681,E2 -20224.681} C_VEL
LIN {X 0,Y 224.83,Z 301.389,A -85,B 0,C 180,E1 -20226.459,E2 -20226.459} C_VEL
LIN {X 0,Y 221.383,Z 307.288,A -85,B 0,C 180,E1 -20229.09,E2 -20229.09} C_VEL
LIN {X 0,Y 220.845,Z 309.286,A -85,B 0,C 180,E1 -20229.997,E2 -20229.997} C_VEL
LIN {X 0,Y 220.476,Z 312.707,A -85,B 0,C 180,E1 -20231.555,E2 -20231.555} C_VEL
LIN {X 0,Y 221.1,Z 332.284,A -85,B 0,C 180,E1 -20232.668,E2 -20232.668} C_VEL
LIN {X 0,Y 222.834,Z 351.785,A -85,B 0,C 180,E1 -20233.749,E2 -20233.749} C_VEL
LIN {X 0,Y 221.932,Z 392.535,A -85,B 0,C 180,E1 -20236.147,E2 -20236.147} C_VEL
LIN {X 0,Y 221.546,Z 405.164,A -85,B 0,C 180,E1 -20237.29,E2 -20237.29} C_VEL
LIN {X 0,Y 221.071,Z 415.326,A -85,B 0,C 180,E1 -20238.543,E2 -20238.543} C_VEL
LIN {X 0,Y 220.586,Z 425.486,A -85,B 0,C 180,E1 -20240.143,E2 -20240.143} C_VEL
LIN {X 0,Y 220.35,Z 434.902,A -85,B 0,C 180,E1 -20242.045,E2 -20242.045} C_VEL
LIN {X 0,Y 220.14,Z 442.903,A -85,B 0,C 180,E1 -20244.048,E2 -20244.048} C_VEL
LIN {X 0,Y 219.951,Z 450.303,A -85,B 0,C 180,E1 -20246.339,E2 -20246.339} C_VEL
LIN {X 0,Y 219.766,Z 457.026,A -85,B 0,C 180,E1 -20249.087,E2 -20249.087} C_VEL
LIN {X 0,Y 219.531,Z 460.554,A -85,B 0,C 180,E1 -20250.92,E2 -20250.92} C_VEL
LIN {X 0,Y 219.123,Z 464.431,A -85,B 0,C 180,E1 -20253.681,E2 -20253.681} C_VEL
LIN {X 0,Y 219.023,Z 466.639,A -85,B 0,C 180,E1 -20255.828,E2 -20255.828} C_VEL
LIN {X 0,Y 219.133,Z 467.827,A -85,B 0,C 180,E1 -20257.374,E2 -20257.374} C_VEL
LIN {X 0,Y 219.492,Z 468.712,A -85,B 0,C 180,E1 -20259.216,E2 -20259.216} C_VEL
LIN {X 0,Y 220.168,Z 469.181,A -85,B 0,C 180,E1 -20261.045,E2 -20261.045} C_VEL
LIN {X 0,Y 221.154,Z 469.247,A -85,B 0,C 180,E1 -20262.856,E2 -20262.856} C_VEL
LIN {X 0,Y 222.419,Z 468.745,A -85,B 0,C 180,E1 -20264.645,E2 -20264.645} C_VEL
LIN {X 0,Y 224.001,Z 467.768,A -85,B 0,C 180,E1 -20266.405,E2 -20266.405} C_VEL
LIN {X 0,Y 225.877,Z 466.386,A -85,B 0,C 180,E1 -20268.131,E2 -20268.131} C_VEL
LIN {X 0,Y 229.001,Z 463.344,A -85,B 0,C 180,E1 -20270.67,E2 -20270.67} C_VEL
LIN {X 0,Y 232.863,Z 459.08,A -85,B 0,C 180,E1 -20273.104,E2 -20273.104} C_VEL
LIN {X 0,Y 237.394,Z 453.555,A -85,B 0,C 180,E1 -20275.424,E2 -20275.424} C_VEL
LIN {X 0,Y 242.417,Z 446.363,A -85,B 0,C 180,E1 -20277.639,E2 -20277.639} C_VEL
LIN {X 0,Y 247,Z 438.935,A -85,B 0,C 180,E1 -20279.397,E2 -20279.397} C_VEL
LIN {X 0,Y 251.034,Z 431.782,A -85,B 0,C 180,E1 -20280.729,E2 -20280.729} C_VEL
LIN {X 0,Y 255.853,Z 422.053,A -85,B 0,C 180,E1 -20282.158,E2 -20282.158} C_VEL
LIN {X 0,Y 260.547,Z 410.683,A -85,B 0,C 180,E1 -20283.411,E2 -20283.411} C_VEL
LIN {X 0,Y 264.842,Z 398.333,A -85,B 0,C 180,E1 -20284.42,E2 -20284.42} C_VEL
LIN {X 0,Y 268.164,Z 385.151,A -85,B 0,C 180,E1 -20285.212,E2 -20285.212} C_VEL
LIN {X 0,Y 270.56,Z 372.58,A -85,B 0,C 180,E1 -20285.861,E2 -20285.861} C_VEL
LIN {X 0,Y 270.615,Z 370.025,A -85,B 0,C 180,E1 -20286.241,E2 -20286.241} C_VEL
LIN {X 0,Y 269.332,Z 365.097,A -85,B 0,C 180,E1 -20287.972,E2 -20287.972} C_VEL
LIN {X 0,Y 268.229,Z 361.277,A -85,B 0,C 180,E1 -20289.804,E2 -20289.804} C_VEL
LIN {X 0,Y 267.157,Z 357.624,A -85,B 0,C 180,E1 -20292.466,E2 -20292.466} C_VEL
LIN {X 0,Y 266.902,Z 356.427,A -85,B 0,C 180,E1 -20293.961,E2 -20293.961} C_VEL
LIN {X 0,Y 266.774,Z 355.926,A -85,B 0,C 180,E1 -20295.343,E2 -20295.343} C_VEL
LIN {X 0,Y 267.227,Z 356.089,A -85,B 0,C 180,E1 -20297.829,E2 -20297.829} C_VEL
LIN {X 0,Y 268.76,Z 358.072,A -85,B 0,C 180,E1 -20300.801,E2 -20300.801} C_VEL
LIN {X 0,Y 270.548,Z 361.821,A -85,B 0,C 180,E1 -20303.183,E2 -20303.183} C_VEL
LIN {X 0,Y 271.73,Z 364.527,A -85,B 0,C 180,E1 -20304.469,E2 -20304.469} C_VEL
LIN {X 0,Y 267.77,Z 384.136,A -85,B 0,C 180,E1 -20305.511,E2 -20305.511} C_VEL
LIN {X 0,Y 264.652,Z 395.12,A -85,B 0,C 180,E1 -20306.327,E2 -20306.327} C_VEL
LIN {X 0,Y 260.886,Z 405.929,A -85,B 0,C 180,E1 -20307.392,E2 -20307.392} C_VEL
LIN {X 0,Y 256.277,Z 416.698,A -85,B 0,C 180,E1 -20308.82,E2 -20308.82} C_VEL
LIN {X 0,Y 251.932,Z 425.422,A -85,B 0,C 180,E1 -20310.312,E2 -20310.312} C_VEL
LIN {X 0,Y 247.341,Z 433.302,A -85,B 0,C 180,E1 -20312.034,E2 -20312.034} C_VEL
LIN {X 0,Y 242.207,Z 440.739,A -85,B 0,C 180,E1 -20314.191,E2 -20314.191} C_VEL
LIN {X 0,Y 238.429,Z 445.577,A -85,B 0,C 180,E1 -20316.036,E2 -20316.036} C_VEL
LIN {X 0,Y 234.801,Z 449.565,A -85,B 0,C 180,E1 -20318.02,E2 -20318.02} C_VEL
LIN {X 0,Y 230.917,Z 453.143,A -85,B 0,C 180,E1 -20320.432,E2 -20320.432} C_VEL
LIN {X 0,Y 228.622,Z 454.784,A -85,B 0,C 180,E1 -20322.089,E2 -20322.089} C_VEL
LIN {X 0,Y 226.479,Z 455.965,A -85,B 0,C 180,E1 -20323.774,E2 -20323.774} C_VEL
LIN {X 0,Y 224.66,Z 456.688,A -85,B 0,C 180,E1 -20325.498,E2 -20325.498} C_VEL
LIN {X 0,Y 223.227,Z 456.839,A -85,B 0,C 180,E1 -20327.26,E2 -20327.26} C_VEL
LIN {X 0,Y 221.815,Z 456.496,A -85,B 0,C 180,E1 -20329.032,E2 -20329.032} C_VEL
LIN {X 0,Y 220.697,Z 455.712,A -85,B 0,C 180,E1 -20330.829,E2 -20330.829} C_VEL
LIN {X 0,Y 219.943,Z 454.493,A -85,B 0,C 180,E1 -20332.648,E2 -20332.648} C_VEL
LIN {X 0,Y 219.297,Z 451.581,A -85,B 0,C 180,E1 -20335.396,E2 -20335.396} C_VEL
LIN {X 0,Y 218.894,Z 447.433,A -85,B 0,C 180,E1 -20338.151,E2 -20338.151} C_VEL
LIN {X 0,Y 218.889,Z 441.958,A -85,B 0,C 180,E1 -20340.911,E2 -20340.911} C_VEL
LIN {X 0,Y 219.202,Z 434.807,A -85,B 0,C 180,E1 -20343.667,E2 -20343.667} C_VEL
LIN {X 0,Y 219.464,Z 427.31,A -85,B 0,C 180,E1 -20345.896,E2 -20345.896} C_VEL
LIN {X 0,Y 219.858,Z 419.537,A -85,B 0,C 180,E1 -20347.797,E2 -20347.797} C_VEL
LIN {X 0,Y 220.271,Z 410.401,A -85,B 0,C 180,E1 -20349.633,E2 -20349.633} C_VEL
LIN {X 0,Y 220.829,Z 400.361,A -85,B 0,C 180,E1 -20351.231,E2 -20351.231} C_VEL
LIN {X 0,Y 221.279,Z 389.281,A -85,B 0,C 180,E1 -20352.602,E2 -20352.602} C_VEL
LIN {X 0,Y 221.821,Z 377.137,A -85,B 0,C 180,E1 -20353.736,E2 -20353.736} C_VEL
LIN {X 0,Y 222.397,Z 353.35,A -85,B 0,C 180,E1 -20355.16,E2 -20355.16} C_VEL
LIN {X 0,Y 223.006,Z 318.496,A -85,B 0,C 180,E1 -20357.118,E2 -20357.118} C_VEL
LIN {X 0,Y 220.947,Z 297.777,A -85,B 0,C 180,E1 -20358.301,E2 -20358.301} C_VEL
LIN {X 0,Y 220.857,Z 297.782,A -85,B 0,C 180,E1 -20362.652,E2 -20362.652} C_VEL
LIN {X 0,Y 220.836,Z 297.787,A -85,B 0,C 180,E1 -20366.985,E2 -20366.985} C_VEL
LIN {X 0,Y 220.805,Z 297.788,A -85,B 0,C 180,E1 -20370.748,E2 -20370.748} C_VEL
LIN {X 0,Y 220.774,Z 297.796,A -85,B 0,C 180,E1 -20374.946,E2 -20374.946} C_VEL
LIN {X 0,Y 220.777,Z 297.794,A -85,B 0,C 180,E1 -20377.263,E2 -20377.263} C_VEL
LIN {X 0,Y 220.723,Z 297.799,A -85,B 0,C 180,E1 -20381.948,E2 -20381.948} C_VEL
LIN {X 0,Y 220.736,Z 297.8,A -85,B 0,C 180,E1 -20385.533,E2 -20385.533} C_VEL
LIN {X 0,Y 220.756,Z 297.795,A -85,B 0,C 180,E1 -20390.449,E2 -20390.449} C_VEL
LIN {X 0,Y 220.795,Z 297.794,A -85,B 0,C 180,E1 -20392.784,E2 -20392.784} C_VEL
LIN {X 0,Y 220.779,Z 297.794,A -85,B 0,C 180,E1 -20397.234,E2 -20397.234} C_VEL
LIN {X 0,Y 220.777,Z 297.797,A -85,B 0,C 180,E1 -20401.475,E2 -20401.475} C_VEL
LIN {X 0,Y 220.823,Z 297.789,A -85,B 0,C 180,E1 -20405.557,E2 -20405.557} C_VEL
LIN {X 0,Y 220.842,Z 297.789,A -85,B 0,C 180,E1 -20409.506,E2 -20409.506} C_VEL
LIN {X 0,Y 220.965,Z 297.774,A -85,B 0,C 180,E1 -20413.363,E2 -20413.363} C_VEL
LIN {X 0,Y 221.044,Z 297.76,A -85,B 0,C 180,E1 -20418.999,E2 -20418.999} C_VEL
LIN {X 0,Y 221.22,Z 297.739,A -85,B 0,C 180,E1 -20422.696,E2 -20422.696} C_VEL
LIN {X 0,Y 221.474,Z 297.71,A -85,B 0,C 180,E1 -20428.178,E2 -20428.178} C_VEL
LIN {X 0,Y 221.473,Z 297.71,A -85,B 0,C 180,E1 -20431.815,E2 -20431.815} C_VEL
LIN {X 0,Y 221.216,Z 297.739,A -85,B 0,C 180,E1 -20437.298,E2 -20437.298} C_VEL
LIN {X 0,Y 221.039,Z 297.761,A -85,B 0,C 180,E1 -20440.995,E2 -20440.995} C_VEL
LIN {X 0,Y 220.958,Z 297.775,A -85,B 0,C 180,E1 -20446.631,E2 -20446.631} C_VEL
LIN {X 0,Y 220.834,Z 297.79,A -85,B 0,C 180,E1 -20450.488,E2 -20450.488} C_VEL
LIN {X 0,Y 220.813,Z 297.79,A -85,B 0,C 180,E1 -20454.438,E2 -20454.438} C_VEL
LIN {X 0,Y 220.789,Z 297.795,A -85,B 0,C 180,E1 -20458.516,E2 -20458.516} C_VEL
LIN {X 0,Y 220.778,Z 297.794,A -85,B 0,C 180,E1 -20462.758,E2 -20462.758} C_VEL
LIN {X 0,Y 220.795,Z 297.794,A -85,B 0,C 180,E1 -20467.292,E2 -20467.292} C_VEL
LIN {X 0,Y 220.831,Z 297.786,A -85,B 0,C 180,E1 -20471.933,E2 -20471.933} C_VEL
LIN {X 0,Y 220.833,Z 297.789,A -85,B 0,C 180,E1 -20475.577,E2 -20475.577} C_VEL
LIN {X 0,Y 220.819,Z 297.788,A -85,B 0,C 180,E1 -20479.799,E2 -20479.799} C_VEL
LIN {X 0,Y 220.797,Z 297.792,A -85,B 0,C 180,E1 -20482.801,E2 -20482.801} C_VEL
LIN {X 0,Y 220.788,Z 297.794,A -85,B 0,C 180,E1 -20487.252,E2 -20487.252} C_VEL
LIN {X 0,Y 220.794,Z 297.794,A -85,B 0,C 180,E1 -20491.493,E2 -20491.493} C_VEL
LIN {X 0,Y 220.831,Z 297.789,A -85,B 0,C 180,E1 -20495.572,E2 -20495.572} C_VEL
LIN {X 0,Y 220.841,Z 297.786,A -85,B 0,C 180,E1 -20499.52,E2 -20499.52} C_VEL
LIN {X 0,Y 220.954,Z 297.773,A -85,B 0,C 180,E1 -20503.376,E2 -20503.376} C_VEL
LIN {X 0,Y 221.041,Z 297.761,A -85,B 0,C 180,E1 -20509.012,E2 -20509.012} C_VEL
LIN {X 0,Y 221.229,Z 297.738,A -85,B 0,C 180,E1 -20512.709,E2 -20512.709} C_VEL
LIN {X 0,Y 221.456,Z 297.711,A -85,B 0,C 180,E1 -20518.191,E2 -20518.191} C_VEL
LIN {X 0,Y 221.459,Z 297.709,A -85,B 0,C 180,E1 -20521.828,E2 -20521.828} C_VEL
LIN {X 0,Y 221.226,Z 297.739,A -85,B 0,C 180,E1 -20527.309,E2 -20527.309} C_VEL
LIN {X 0,Y 221.05,Z 297.761,A -85,B 0,C 180,E1 -20531.006,E2 -20531.006} C_VEL
LIN {X 0,Y 220.96,Z 297.773,A -85,B 0,C 180,E1 -20536.643,E2 -20536.643} C_VEL
LIN {X 0,Y 220.842,Z 297.786,A -85,B 0,C 180,E1 -20540.5,E2 -20540.5} C_VEL
LIN {X 0,Y 220.795,Z 297.791,A -85,B 0,C 180,E1 -20544.452,E2 -20544.452} C_VEL
LIN {X 0,Y 220.799,Z 297.792,A -85,B 0,C 180,E1 -20548.527,E2 -20548.527} C_VEL
LIN {X 0,Y 220.814,Z 297.788,A -85,B 0,C 180,E1 -20552.765,E2 -20552.765} C_VEL
LIN {X 0,Y 220.806,Z 297.793,A -85,B 0,C 180,E1 -20557.283,E2 -20557.283} C_VEL
LIN {X 0,Y 220.754,Z 297.798,A -85,B 0,C 180,E1 -20561.966,E2 -20561.966} C_VEL
LIN {X 0,Y 220.76,Z 297.799,A -85,B 0,C 180,E1 -20565.548,E2 -20565.548} C_VEL
LIN {X 0,Y 220.791,Z 297.791,A -85,B 0,C 180,E1 -20570.464,E2 -20570.464} C_VEL
LIN {X 0,Y 220.837,Z 297.787,A -85,B 0,C 180,E1 -20572.8,E2 -20572.8} C_VEL
LIN {X 0,Y 220.824,Z 297.787,A -85,B 0,C 180,E1 -20577.249,E2 -20577.249} C_VEL
LIN {X 0,Y 220.883,Z 297.781,A -85,B 0,C 180,E1 -20581.497,E2 -20581.497} C_VEL
LIN {X 0,Y 221.338,Z 297.849,A -85,B 0,C 180,E1 -20584.81,E2 -20584.81} C_VEL
LIN {X 0,Y 221.941,Z 301.315,A -85,B 0,C 180,E1 -20586.396,E2 -20586.396} C_VEL
LIN {X 0,Y 220.845,Z 309.286,A -85,B 0,C 180,E1 -20589.997,E2 -20589.997} C_VEL
LIN {X 0,Y 220.233,Z 311.64,A -85,B 0,C 180,E1 -20590.756,E2 -20590.756} C_VEL
LIN {X 0,Y 218.831,Z 315.418,A -85,B 0,C 180,E1 -20591.45,E2 -20591.45} C_VEL
LIN {X 0,Y 216.531,Z 321.761,A -85,B 0,C 180,E1 -20592.096,E2 -20592.096} C_VEL
LIN {X 0,Y 214.605,Z 329.392,A -85,B 0,C 180,E1 -20592.554,E2 -20592.554} C_VEL
LIN {X 0,Y 214.319,Z 333.435,A -85,B 0,C 180,E1 -20592.789,E2 -20592.789} C_VEL
LIN {X 0,Y 214.46,Z 337.489,A -85,B 0,C 180,E1 -20593.029,E2 -20593.029} C_VEL
LIN {X 0,Y 215.745,Z 352.046,A -85,B 0,C 180,E1 -20593.868,E2 -20593.868} C_VEL
LIN {X 0,Y 214.899,Z 392.031,A -85,B 0,C 180,E1 -20596.348,E2 -20596.348} C_VEL
LIN {X 0,Y 214.572,Z 404.095,A -85,B 0,C 180,E1 -20597.471,E2 -20597.471} C_VEL
LIN {X 0,Y 214.143,Z 413.458,A -85,B 0,C 180,E1 -20598.647,E2 -20598.647} C_VEL
LIN {X 0,Y 213.718,Z 422.497,A -85,B 0,C 180,E1 -20600.062,E2 -20600.062} C_VEL
LIN {X 0,Y 213.424,Z 432.998,A -85,B 0,C 180,E1 -20602.11,E2 -20602.11} C_VEL
LIN {X 0,Y 213.229,Z 441.785,A -85,B 0,C 180,E1 -20604.329,E2 -20604.329} C_VEL
LIN {X 0,Y 213.101,Z 447.916,A -85,B 0,C 180,E1 -20606.221,E2 -20606.221} C_VEL
LIN {X 0,Y 212.918,Z 452.913,A -85,B 0,C 180,E1 -20608.112,E2 -20608.112} C_VEL
LIN {X 0,Y 212.852,Z 457.058,A -85,B 0,C 180,E1 -20610.003,E2 -20610.003} C_VEL
LIN {X 0,Y 212.281,Z 461.789,A -85,B 0,C 180,E1 -20612.85,E2 -20612.85} C_VEL
LIN {X 0,Y 212.044,Z 465.242,A -85,B 0,C 180,E1 -20615.71,E2 -20615.71} C_VEL
LIN {X 0,Y 212.172,Z 466.812,A -85,B 0,C 180,E1 -20617.617,E2 -20617.617} C_VEL
LIN {X 0,Y 212.519,Z 467.962,A -85,B 0,C 180,E1 -20619.521,E2 -20619.521} C_VEL
LIN {X 0,Y 213.225,Z 468.693,A -85,B 0,C 180,E1 -20621.409,E2 -20621.409} C_VEL
LIN {X 0,Y 214.25,Z 468.859,A -85,B 0,C 180,E1 -20623.278,E2 -20623.278} C_VEL
LIN {X 0,Y 215.568,Z 468.6,A -85,B 0,C 180,E1 -20625.122,E2 -20625.122} C_VEL
LIN {X 0,Y 217.217,Z 467.951,A -85,B 0,C 180,E1 -20626.932,E2 -20626.932} C_VEL
LIN {X 0,Y 219.15,Z 466.792,A -85,B 0,C 180,E1 -20628.708,E2 -20628.708} C_VEL
LIN {X 0,Y 222.441,Z 464.157,A -85,B 0,C 180,E1 -20631.308,E2 -20631.308} C_VEL
LIN {X 0,Y 226.442,Z 460.362,A -85,B 0,C 180,E1 -20633.799,E2 -20633.799} C_VEL
LIN {X 0,Y 231.115,Z 455.218,A -85,B 0,C 180,E1 -20636.166,E2 -20636.166} C_VEL
LIN {X 0,Y 235.415,Z 449.899,A -85,B 0,C 180,E1 -20638.05,E2 -20638.05} C_VEL
LIN {X 0,Y 240.118,Z 443.411,A -85,B 0,C 180,E1 -20639.842,E2 -20639.842} C_VEL
LIN {X 0,Y 245.185,Z 435.485,A -85,B 0,C 180,E1 -20641.544,E2 -20641.544} C_VEL
LIN {X 0,Y 250.705,Z 425.593,A -85,B 0,C 180,E1 -20643.14,E2 -20643.14} C_VEL
LIN {X 0,Y 254.947,Z 416.794,A -85,B 0,C 180,E1 -20644.235,E2 -20644.235} C_VEL
LIN {X 0,Y 259.336,Z 406.173,A -85,B 0,C 180,E1 -20645.258,E2 -20645.258} C_VEL
LIN {X 0,Y 263.356,Z 393.866,A -85,B 0,C 180,E1 -20646.153,E2 -20646.153} C_VEL
LIN {X 0,Y 266.645,Z 380.807,A -85,B 0,C 180,E1 -20646.866,E2 -20646.866} C_VEL
LIN {X 0,Y 267.782,Z 374.872,A -85,B 0,C 180,E1 -20647.193,E2 -20647.193} C_VEL
LIN {X 0,Y 266.823,Z 370.94,A -85,B 0,C 180,E1 -20648.676,E2 -20648.676} C_VEL
LIN {X 0,Y 265.932,Z 367.369,A -85,B 0,C 180,E1 -20650.432,E2 -20650.432} C_VEL
LIN {X 0,Y 265.122,Z 364.041,A -85,B 0,C 180,E1 -20652.998,E2 -20652.998} C_VEL
LIN {X 0,Y 264.972,Z 362.953,A -85,B 0,C 180,E1 -20654.744,E2 -20654.744} C_VEL
LIN {X 0,Y 265.227,Z 362.775,A -85,B 0,C 180,E1 -20657.213,E2 -20657.213} C_VEL
LIN {X 0,Y 266.535,Z 364.463,A -85,B 0,C 180,E1 -20660.306,E2 -20660.306} C_VEL
LIN {X 0,Y 268.209,Z 368.301,A -85,B 0,C 180,E1 -20662.799,E2 -20662.799} C_VEL
LIN {X 0,Y 268.622,Z 369.284,A -85,B 0,C 180,E1 -20663.279,E2 -20663.279} C_VEL
LIN {X 0,Y 265.058,Z 385.138,A -85,B 0,C 180,E1 -20664.114,E2 -20664.114} C_VEL
LIN {X 0,Y 261.89,Z 395.514,A -85,B 0,C 180,E1 -20664.887,E2 -20664.887} C_VEL
LIN {X 0,Y 257.696,Z 406.935,A -85,B 0,C 180,E1 -20666,E2 -20666} C_VEL
LIN {X 0,Y 253.353,Z 416.482,A -85,B 0,C 180,E1 -20667.246,E2 -20667.246} C_VEL
LIN {X 0,Y 249.214,Z 424.286,A -85,B 0,C 180,E1 -20668.545,E2 -20668.545} C_VEL
LIN {X 0,Y 244.309,Z 432.411,A -85,B 0,C 180,E1 -20670.242,E2 -20670.242} C_VEL
LIN {X 0,Y 238.747,Z 440.161,A -85,B 0,C 180,E1 -20672.37,E2 -20672.37} C_VEL
LIN {X 0,Y 234.482,Z 445.217,A -85,B 0,C 180,E1 -20674.232,E2 -20674.232} C_VEL
LIN {X 0,Y 229.863,Z 450.015,A -85,B 0,C 180,E1 -20676.572,E2 -20676.572} C_VEL
LIN {X 0,Y 226.985,Z 452.485,A -85,B 0,C 180,E1 -20678.181,E2 -20678.181} C_VEL
LIN {X 0,Y 224.345,Z 454.439,A -85,B 0,C 180,E1 -20679.835,E2 -20679.835} C_VEL
LIN {X 0,Y 221.963,Z 455.874,A -85,B 0,C 180,E1 -20681.532,E2 -20681.532} C_VEL
LIN {X 0,Y 219.732,Z 456.748,A -85,B 0,C 180,E1 -20683.261,E2 -20683.261} C_VEL
LIN {X 0,Y 217.819,Z 457.161,A -85,B 0,C 180,E1 -20685.033,E2 -20685.033} C_VEL
LIN {X 0,Y 216.326,Z 457.147,A -85,B 0,C 180,E1 -20686.846,E2 -20686.846} C_VEL
LIN {X 0,Y 214.852,Z 456.635,A -85,B 0,C 180,E1 -20688.672,E2 -20688.672} C_VEL
LIN {X 0,Y 213.508,Z 455.296,A -85,B 0,C 180,E1 -20690.948,E2 -20690.948} C_VEL
LIN {X 0,Y 212.437,Z 452.089,A -85,B 0,C 180,E1 -20694.295,E2 -20694.295} C_VEL
LIN {X 0,Y 212.096,Z 449.609,A -85,B 0,C 180,E1 -20696.191,E2 -20696.191} C_VEL
LIN {X 0,Y 211.838,Z 444.619,A -85,B 0,C 180,E1 -20699.04,E2 -20699.04} C_VEL
LIN {X 0,Y 211.978,Z 439.348,A -85,B 0,C 180,E1 -20701.415,E2 -20701.415} C_VEL
LIN {X 0,Y 212.201,Z 434.268,A -85,B 0,C 180,E1 -20703.313,E2 -20703.313} C_VEL
LIN {X 0,Y 212.352,Z 428.168,A -85,B 0,C 180,E1 -20705.212,E2 -20705.212} C_VEL
LIN {X 0,Y 212.763,Z 420.948,A -85,B 0,C 180,E1 -20707.095,E2 -20707.095} C_VEL
LIN {X 0,Y 213.173,Z 412.225,A -85,B 0,C 180,E1 -20708.952,E2 -20708.952} C_VEL
LIN {X 0,Y 213.764,Z 400.774,A -85,B 0,C 180,E1 -20710.887,E2 -20710.887} C_VEL
LIN {X 0,Y 214.239,Z 389.77,A -85,B 0,C 180,E1 -20712.301,E2 -20712.301} C_VEL
LIN {X 0,Y 214.74,Z 377.739,A -85,B 0,C 180,E1 -20713.474,E2 -20713.474} C_VEL
LIN {X 0,Y 215.285,Z 354.49,A -85,B 0,C 180,E1 -20714.947,E2 -20714.947} C_VEL
LIN {X 0,Y 215.956,Z 319.134,A -85,B 0,C 180,E1 -20717.051,E2 -20717.051} C_VEL
LIN {X 0,Y 213.874,Z 298.658,A -85,B 0,C 180,E1 -20718.231,E2 -20718.231} C_VEL
LIN {X 0,Y 213.79,Z 298.661,A -85,B 0,C 180,E1 -20723.222,E2 -20723.222} C_VEL
LIN {X 0,Y 213.774,Z 298.667,A -85,B 0,C 180,E1 -20727.416,E2 -20727.416} C_VEL
LIN {X 0,Y 213.744,Z 298.667,A -85,B 0,C 180,E1 -20731.728,E2 -20731.728} C_VEL
LIN {X 0,Y 213.723,Z 298.676,A -85,B 0,C 180,E1 -20736.278,E2 -20736.278} C_VEL
LIN {X 0,Y 213.674,Z 298.678,A -85,B 0,C 180,E1 -20741.119,E2 -20741.119} C_VEL
LIN {X 0,Y 213.678,Z 298.678,A -85,B 0,C 180,E1 -20743.67,E2 -20743.67} C_VEL
LIN {X 0,Y 213.677,Z 298.68,A -85,B 0,C 180,E1 -20746.335,E2 -20746.335} C_VEL
LIN {X 0,Y 213.68,Z 298.677,A -85,B 0,C 180,E1 -20749.136,E2 -20749.136} C_VEL
LIN {X 0,Y 213.71,Z 298.675,A -85,B 0,C 180,E1 -20753.702,E2 -20753.702} C_VEL
LIN {X 0,Y 213.725,Z 298.669,A -85,B 0,C 180,E1 -20758.252,E2 -20758.252} C_VEL
LIN {X 0,Y 213.791,Z 298.665,A -85,B 0,C 180,E1 -20762.595,E2 -20762.595} C_VEL
LIN {X 0,Y 213.78,Z 298.665,A -85,B 0,C 180,E1 -20766.967,E2 -20766.967} C_VEL
LIN {X 0,Y 213.896,Z 298.652,A -85,B 0,C 180,E1 -20772.797,E2 -20772.797} C_VEL
LIN {X 0,Y 213.903,Z 298.646,A -85,B 0,C 180,E1 -20776.7,E2 -20776.7} C_VEL
LIN {X 0,Y 214.106,Z 298.625,A -85,B 0,C 180,E1 -20780.551,E2 -20780.551} C_VEL
LIN {X 0,Y 214.06,Z 298.629,A -85,B 0,C 180,E1 -20784.344,E2 -20784.344} C_VEL
LIN {X 0,Y 214.432,Z 298.587,A -85,B 0,C 180,E1 -20788.119,E2 -20788.119} C_VEL
LIN {X 0,Y 214.431,Z 298.588,A -85,B 0,C 180,E1 -20791.875,E2 -20791.875} C_VEL
LIN {X 0,Y 214.156,Z 298.619,A -85,B 0,C 180,E1 -20797.54,E2 -20797.54} C_VEL
LIN {X 0,Y 213.962,Z 298.642,A -85,B 0,C 180,E1 -20801.363,E2 -20801.363} C_VEL
LIN {X 0,Y 213.872,Z 298.653,A -85,B 0,C 180,E1 -20805.238,E2 -20805.238} C_VEL
LIN {X 0,Y 213.784,Z 298.665,A -85,B 0,C 180,E1 -20809.189,E2 -20809.189} C_VEL
LIN {X 0,Y 213.763,Z 298.666,A -85,B 0,C 180,E1 -20813.233,E2 -20813.233} C_VEL
LIN {X 0,Y 213.783,Z 298.666,A -85,B 0,C 180,E1 -20817.452,E2 -20817.452} C_VEL
LIN {X 0,Y 213.733,Z 298.668,A -85,B 0,C 180,E1 -20821.739,E2 -20821.739} C_VEL
LIN {X 0,Y 213.71,Z 298.675,A -85,B 0,C 180,E1 -20826.29,E2 -20826.29} C_VEL
LIN {X 0,Y 213.782,Z 298.665,A -85,B 0,C 180,E1 -20831.104,E2 -20831.104} C_VEL
LIN {X 0,Y 213.795,Z 298.665,A -85,B 0,C 180,E1 -20833.698,E2 -20833.698} C_VEL
LIN {X 0,Y 213.801,Z 298.663,A -85,B 0,C 180,E1 -20836.362,E2 -20836.362} C_VEL
LIN {X 0,Y 213.746,Z 298.671,A -85,B 0,C 180,E1 -20841.353,E2 -20841.353} C_VEL
LIN {X 0,Y 213.733,Z 298.672,A -85,B 0,C 180,E1 -20846.027,E2 -20846.027} C_VEL
LIN {X 0,Y 213.727,Z 298.672,A -85,B 0,C 180,E1 -20850.459,E2 -20850.459} C_VEL
LIN {X 0,Y 213.767,Z 298.667,A -85,B 0,C 180,E1 -20854.709,E2 -20854.709} C_VEL
LIN {X 0,Y 213.764,Z 298.666,A -85,B 0,C 180,E1 -20858.81,E2 -20858.81} C_VEL
LIN {X 0,Y 213.867,Z 298.655,A -85,B 0,C 180,E1 -20862.808,E2 -20862.808} C_VEL
LIN {X 0,Y 213.912,Z 298.647,A -85,B 0,C 180,E1 -20866.714,E2 -20866.714} C_VEL
LIN {X 0,Y 214.117,Z 298.626,A -85,B 0,C 180,E1 -20870.564,E2 -20870.564} C_VEL
LIN {X 0,Y 214.064,Z 298.631,A -85,B 0,C 180,E1 -20874.357,E2 -20874.357} C_VEL
LIN {X 0,Y 214.393,Z 298.59,A -85,B 0,C 180,E1 -20878.131,E2 -20878.131} C_VEL
LIN {X 0,Y 214.498,Z 298.578,A -85,B 0,C 180,E1 -20880.009,E2 -20880.009} C_VEL
LIN {X 0,Y 214.396,Z 298.589,A -85,B 0,C 180,E1 -20881.888,E2 -20881.888} C_VEL
LIN {X 0,Y 214.167,Z 298.618,A -85,B 0,C 180,E1 -20887.552,E2 -20887.552} C_VEL
LIN {X 0,Y 213.98,Z 298.64,A -85,B 0,C 180,E1 -20891.374,E2 -20891.374} C_VEL
LIN {X 0,Y 213.862,Z 298.657,A -85,B 0,C 180,E1 -20895.251,E2 -20895.251} C_VEL
LIN {X 0,Y 213.786,Z 298.667,A -85,B 0,C 180,E1 -20899.201,E2 -20899.201} C_VEL
LIN {X 0,Y 213.762,Z 298.668,A -85,B 0,C 180,E1 -20903.246,E2 -20903.246} C_VEL
LIN {X 0,Y 213.786,Z 298.668,A -85,B 0,C 180,E1 -20907.435,E2 -20907.435} C_VEL
LIN {X 0,Y 213.761,Z 298.667,A -85,B 0,C 180,E1 -20911.748,E2 -20911.748} C_VEL
LIN {X 0,Y 213.746,Z 298.67,A -85,B 0,C 180,E1 -20916.297,E2 -20916.297} C_VEL
LIN {X 0,Y 213.704,Z 298.672,A -85,B 0,C 180,E1 -20921.137,E2 -20921.137} C_VEL
LIN {X 0,Y 213.709,Z 298.678,A -85,B 0,C 180,E1 -20923.688,E2 -20923.688} C_VEL
LIN {X 0,Y 213.71,Z 298.675,A -85,B 0,C 180,E1 -20926.353,E2 -20926.353} C_VEL
LIN {X 0,Y 213.714,Z 298.673,A -85,B 0,C 180,E1 -20931.336,E2 -20931.336} C_VEL
LIN {X 0,Y 213.766,Z 298.67,A -85,B 0,C 180,E1 -20936.024,E2 -20936.024} C_VEL
LIN {X 0,Y 213.793,Z 298.666,A -85,B 0,C 180,E1 -20940.46,E2 -20940.46} C_VEL
LIN {X 0,Y 214.384,Z 298.798,A -85,B 0,C 180,E1 -20945.14,E2 -20945.14} C_VEL
LIN {X 0,Y 214.826,Z 301.406,A -85,B 0,C 180,E1 -20946.367,E2 -20946.367} C_VEL
LIN {X 0,Y 213.368,Z 312.411,A -85,B 0,C 180,E1 -20951.54,E2 -20951.54} C_VEL
LIN {X 0,Y 213.97,Z 331.848,A -85,B 0,C 180,E1 -20952.705,E2 -20952.705} C_VEL
LIN {X 0,Y 214.46,Z 337.489,A -85,B 0,C 180,E1 -20953.029,E2 -20953.029} C_VEL
LIN {X 0,Y 214.122,Z 343.255,A -85,B 0,C 180,E1 -20953.372,E2 -20953.372} C_VEL
LIN {X 0,Y 211.631,Z 352.604,A -85,B 0,C 180,E1 -20953.994,E2 -20953.994} C_VEL
LIN {X 0,Y 208.954,Z 361.95,A -85,B 0,C 180,E1 -20954.642,E2 -20954.642} C_VEL
LIN {X 0,Y 208.351,Z 367.723,A -85,B 0,C 180,E1 -20955.021,E2 -20955.021} C_VEL
LIN {X 0,Y 207.856,Z 392.801,A -85,B 0,C 180,E1 -20956.686,E2 -20956.686} C_VEL
LIN {X 0,Y 207.554,Z 403.923,A -85,B 0,C 180,E1 -20957.786,E2 -20957.786} C_VEL
LIN {X 0,Y 207.146,Z 413.247,A -85,B 0,C 180,E1 -20959.001,E2 -20959.001} C_VEL
LIN {X 0,Y 206.738,Z 422.556,A -85,B 0,C 180,E1 -20960.516,E2 -20960.516} C_VEL
LIN {X 0,Y 206.494,Z 432.051,A -85,B 0,C 180,E1 -20962.425,E2 -20962.425} C_VEL
LIN {X 0,Y 206.346,Z 440.558,A -85,B 0,C 180,E1 -20964.629,E2 -20964.629} C_VEL
LIN {X 0,Y 206.215,Z 446.735,A -85,B 0,C 180,E1 -20966.584,E2 -20966.584} C_VEL
LIN {X 0,Y 206.018,Z 452.967,A -85,B 0,C 180,E1 -20969.026,E2 -20969.026} C_VEL
LIN {X 0,Y 205.803,Z 456.976,A -85,B 0,C 180,E1 -20970.982,E2 -20970.982} C_VEL
LIN {X 0,Y 205.235,Z 461.589,A -85,B 0,C 180,E1 -20973.93,E2 -20973.93} C_VEL
LIN {X 0,Y 205.093,Z 464.348,A -85,B 0,C 180,E1 -20976.348,E2 -20976.348} C_VEL
LIN {X 0,Y 205.558,Z 467.129,A -85,B 0,C 180,E1 -20979.846,E2 -20979.846} C_VEL
LIN {X 0,Y 206.297,Z 467.961,A -85,B 0,C 180,E1 -20981.798,E2 -20981.798} C_VEL
LIN {X 0,Y 208.738,Z 468.451,A -85,B 0,C 180,E1 -20985.629,E2 -20985.629} C_VEL
LIN {X 0,Y 210.433,Z 467.945,A -85,B 0,C 180,E1 -20987.496,E2 -20987.496} C_VEL
LIN {X 0,Y 214.598,Z 465.658,A -85,B 0,C 180,E1 -20991.118,E2 -20991.118} C_VEL
LIN {X 0,Y 218.6,Z 462.658,A -85,B 0,C 180,E1 -20993.698,E2 -20993.698} C_VEL
LIN {X 0,Y 223.203,Z 458.507,A -85,B 0,C 180,E1 -20996.159,E2 -20996.159} C_VEL
LIN {X 0,Y 228.413,Z 453.095,A -85,B 0,C 180,E1 -20998.487,E2 -20998.487} C_VEL
LIN {X 0,Y 234.193,Z 446.126,A -85,B 0,C 180,E1 -21000.677,E2 -21000.677} C_VEL
LIN {X 0,Y 239.421,Z 438.909,A -85,B 0,C 180,E1 -21002.395,E2 -21002.395} C_VEL
LIN {X 0,Y 243.886,Z 431.961,A -85,B 0,C 180,E1 -21003.694,E2 -21003.694} C_VEL
LIN {X 0,Y 249.229,Z 422.494,A -85,B 0,C 180,E1 -21005.071,E2 -21005.071} C_VEL
LIN {X 0,Y 254.606,Z 411.386,A -85,B 0,C 180,E1 -21006.297,E2 -21006.297} C_VEL
LIN {X 0,Y 258.823,Z 400.675,A -85,B 0,C 180,E1 -21007.175,E2 -21007.175} C_VEL
LIN {X 0,Y 262.731,Z 388.104,A -85,B 0,C 180,E1 -21007.972,E2 -21007.972} C_VEL
LIN {X 0,Y 264.863,Z 379.116,A -85,B 0,C 180,E1 -21008.435,E2 -21008.435} C_VEL
LIN {X 0,Y 263.978,Z 374.499,A -85,B 0,C 180,E1 -21010.442,E2 -21010.442} C_VEL
LIN {X 0,Y 263.228,Z 371.039,A -85,B 0,C 180,E1 -21013.012,E2 -21013.012} C_VEL
LIN {X 0,Y 263.153,Z 369.99,A -85,B 0,C 180,E1 -21014.343,E2 -21014.343} C_VEL
LIN {X 0,Y 263.342,Z 369.603,A -85,B 0,C 180,E1 -21017.021,E2 -21017.021} C_VEL
LIN {X 0,Y 264.387,Z 371.034,A -85,B 0,C 180,E1 -21019.866,E2 -21019.866} C_VEL
LIN {X 0,Y 265.655,Z 374.076,A -85,B 0,C 180,E1 -21022.023,E2 -21022.023} C_VEL
LIN {X 0,Y 262.413,Z 386.953,A -85,B 0,C 180,E1 -21022.738,E2 -21022.738} C_VEL
LIN {X 0,Y 259.45,Z 396.201,A -85,B 0,C 180,E1 -21023.413,E2 -21023.413} C_VEL
LIN {X 0,Y 255.313,Z 406.835,A -85,B 0,C 180,E1 -21024.436,E2 -21024.436} C_VEL
LIN {X 0,Y 250.675,Z 416.433,A -85,B 0,C 180,E1 -21025.644,E2 -21025.644} C_VEL
LIN {X 0,Y 245.781,Z 425.176,A -85,B 0,C 180,E1 -21027.084,E2 -21027.084} C_VEL
LIN {X 0,Y 240.58,Z 433.191,A -85,B 0,C 180,E1 -21028.759,E2 -21028.759} C_VEL
LIN {X 0,Y 234.634,Z 440.761,A -85,B 0,C 180,E1 -21030.866,E2 -21030.866} C_VEL
LIN {X 0,Y 230.099,Z 445.813,A -85,B 0,C 180,E1 -21032.724,E2 -21032.724} C_VEL
LIN {X 0,Y 226.732,Z 449.124,A -85,B 0,C 180,E1 -21034.273,E2 -21034.273} C_VEL
LIN {X 0,Y 223.544,Z 451.852,A -85,B 0,C 180,E1 -21035.868,E2 -21035.868} C_VEL
LIN {X 0,Y 220.543,Z 453.993,A -85,B 0,C 180,E1 -21037.509,E2 -21037.509} C_VEL
LIN {X 0,Y 217.792,Z 455.602,A -85,B 0,C 180,E1 -21039.2,E2 -21039.2} C_VEL
LIN {X 0,Y 215.3,Z 456.752,A -85,B 0,C 180,E1 -21040.939,E2 -21040.939} C_VEL
LIN {X 0,Y 212.986,Z 457.47,A -85,B 0,C 180,E1 -21042.715,E2 -21042.715} C_VEL
LIN {X 0,Y 211.01,Z 457.621,A -85,B 0,C 180,E1 -21044.538,E2 -21044.538} C_VEL
LIN {X 0,Y 209.439,Z 457.284,A -85,B 0,C 180,E1 -21046.405,E2 -21046.405} C_VEL
LIN {X 0,Y 207.909,Z 456.538,A -85,B 0,C 180,E1 -21048.289,E2 -21048.289} C_VEL
LIN {X 0,Y 206.388,Z 454.686,A -85,B 0,C 180,E1 -21050.953,E2 -21050.953} C_VEL
LIN {X 0,Y 205.724,Z 452.97,A -85,B 0,C 180,E1 -21052.761,E2 -21052.761} C_VEL
LIN {X 0,Y 205.11,Z 448.555,A -85,B 0,C 180,E1 -21056.061,E2 -21056.061} C_VEL
LIN {X 0,Y 204.861,Z 443.272,A -85,B 0,C 180,E1 -21059.007,E2 -21059.007} C_VEL
LIN {X 0,Y 205.024,Z 437.683,A -85,B 0,C 180,E1 -21061.463,E2 -21061.463} C_VEL
LIN {X 0,Y 205.277,Z 430.76,A -85,B 0,C 180,E1 -21063.916,E2 -21063.916} C_VEL
LIN {X 0,Y 205.684,Z 422.041,A -85,B 0,C 180,E1 -21066.354,E2 -21066.354} C_VEL
LIN {X 0,Y 206.058,Z 413.657,A -85,B 0,C 180,E1 -21068.262,E2 -21068.262} C_VEL
LIN {X 0,Y 206.497,Z 404.156,A -85,B 0,C 180,E1 -21070.035,E2 -21070.035} C_VEL
LIN {X 0,Y 207.014,Z 393.276,A -85,B 0,C 180,E1 -21071.618,E2 -21071.618} C_VEL
LIN {X 0,Y 207.532,Z 382.219,A -85,B 0,C 180,E1 -21072.83,E2 -21072.83} C_VEL
LIN {X 0,Y 207.876,Z 369.995,A -85,B 0,C 180,E1 -21073.803,E2 -21073.803} C_VEL
LIN {X 0,Y 208.902,Z 319.852,A -85,B 0,C 180,E1 -21076.92,E2 -21076.92} C_VEL
LIN {X 0,Y 206.861,Z 299.698,A -85,B 0,C 180,E1 -21078.132,E2 -21078.132} C_VEL
LIN {X 0,Y 206.743,Z 299.542,A -85,B 0,C 180,E1 -21081.946,E2 -21081.946} C_VEL
LIN {X 0,Y 206.682,Z 299.554,A -85,B 0,C 180,E1 -21086.222,E2 -21086.222} C_VEL
LIN {X 0,Y 206.681,Z 299.548,A -85,B 0,C 180,E1 -21090.655,E2 -21090.655} C_VEL
LIN {X 0,Y 206.683,Z 299.55,A -85,B 0,C 180,E1 -21095.3,E2 -21095.3} C_VEL
LIN {X 0,Y 206.624,Z 299.556,A -85,B 0,C 180,E1 -21100.244,E2 -21100.244} C_VEL
LIN {X 0,Y 206.606,Z 299.561,A -85,B 0,C 180,E1 -21104.407,E2 -21104.407} C_VEL
LIN {X 0,Y 206.608,Z 299.559,A -85,B 0,C 180,E1 -21108.429,E2 -21108.429} C_VEL
LIN {X 0,Y 206.639,Z 299.555,A -85,B 0,C 180,E1 -21112.248,E2 -21112.248} C_VEL
LIN {X 0,Y 206.661,Z 299.553,A -85,B 0,C 180,E1 -21117.032,E2 -21117.032} C_VEL
LIN {X 0,Y 206.717,Z 299.546,A -85,B 0,C 180,E1 -21122.096,E2 -21122.096} C_VEL
LIN {X 0,Y 206.715,Z 299.544,A -85,B 0,C 180,E1 -21126.597,E2 -21126.597} C_VEL
LIN {X 0,Y 206.827,Z 299.533,A -85,B 0,C 180,E1 -21132.189,E2 -21132.189} C_VEL
LIN {X 0,Y 206.845,Z 299.526,A -85,B 0,C 180,E1 -21136.238,E2 -21136.238} C_VEL
LIN {X 0,Y 207.076,Z 299.502,A -85,B 0,C 180,E1 -21140.227,E2 -21140.227} C_VEL
LIN {X 0,Y 207.021,Z 299.506,A -85,B 0,C 180,E1 -21144.151,E2 -21144.151} C_VEL
LIN {X 0,Y 207.365,Z 299.468,A -85,B 0,C 180,E1 -21148.055,E2 -21148.055} C_VEL
LIN {X 0,Y 207.472,Z 299.456,A -85,B 0,C 180,E1 -21149.997,E2 -21149.997} C_VEL
LIN {X 0,Y 207.364,Z 299.468,A -85,B 0,C 180,E1 -21151.939,E2 -21151.939} C_VEL
LIN {X 0,Y 207.099,Z 299.499,A -85,B 0,C 180,E1 -21157.798,E2 -21157.798} C_VEL
LIN {X 0,Y 207.028,Z 299.511,A -85,B 0,C 180,E1 -21160.185,E2 -21160.185} C_VEL
LIN {X 0,Y 206.807,Z 299.534,A -85,B 0,C 180,E1 -21165.772,E2 -21165.772} C_VEL
LIN {X 0,Y 206.712,Z 299.546,A -85,B 0,C 180,E1 -21169.872,E2 -21169.872} C_VEL
LIN {X 0,Y 206.699,Z 299.546,A -85,B 0,C 180,E1 -21174.076,E2 -21174.076} C_VEL
LIN {X 0,Y 206.698,Z 299.55,A -85,B 0,C 180,E1 -21178.421,E2 -21178.421} C_VEL
LIN {X 0,Y 206.663,Z 299.553,A -85,B 0,C 180,E1 -21182.96,E2 -21182.96} C_VEL
LIN {X 0,Y 206.682,Z 299.55,A -85,B 0,C 180,E1 -21187.734,E2 -21187.734} C_VEL
LIN {X 0,Y 206.707,Z 299.546,A -85,B 0,C 180,E1 -21191.602,E2 -21191.602} C_VEL
LIN {X 0,Y 206.706,Z 299.549,A -85,B 0,C 180,E1 -21195.556,E2 -21195.556} C_VEL
LIN {X 0,Y 206.69,Z 299.548,A -85,B 0,C 180,E1 -21199.771,E2 -21199.771} C_VEL
LIN {X 0,Y 206.689,Z 299.549,A -85,B 0,C 180,E1 -21202.277,E2 -21202.277} C_VEL
LIN {X 0,Y 206.671,Z 299.551,A -85,B 0,C 180,E1 -21207.051,E2 -21207.051} C_VEL
LIN {X 0,Y 206.733,Z 299.546,A -85,B 0,C 180,E1 -21212.106,E2 -21212.106} C_VEL
LIN {X 0,Y 206.724,Z 299.542,A -85,B 0,C 180,E1 -21216.613,E2 -21216.613} C_VEL
LIN {X 0,Y 206.799,Z 299.538,A -85,B 0,C 180,E1 -21222.201,E2 -21222.201} C_VEL
LIN {X 0,Y 206.853,Z 299.528,A -85,B 0,C 180,E1 -21226.252,E2 -21226.252} C_VEL
LIN {X 0,Y 207.079,Z 299.504,A -85,B 0,C 180,E1 -21230.24,E2 -21230.24} C_VEL
LIN {X 0,Y 207.027,Z 299.508,A -85,B 0,C 180,E1 -21234.165,E2 -21234.165} C_VEL
LIN {X 0,Y 207.332,Z 299.469,A -85,B 0,C 180,E1 -21238.067,E2 -21238.067} C_VEL
LIN {X 0,Y 207.466,Z 299.454,A -85,B 0,C 180,E1 -21240.01,E2 -21240.01} C_VEL
LIN {X 0,Y 207.335,Z 299.469,A -85,B 0,C 180,E1 -21241.952,E2 -21241.952} C_VEL
LIN {X 0,Y 207.112,Z 299.496,A -85,B 0,C 180,E1 -21247.81,E2 -21247.81} C_VEL
LIN {X 0,Y 206.899,Z 299.521,A -85,B 0,C 180,E1 -21251.769,E2 -21251.769} C_VEL
LIN {X 0,Y 206.795,Z 299.535,A -85,B 0,C 180,E1 -21255.786,E2 -21255.786} C_VEL
LIN {X 0,Y 206.707,Z 299.546,A -85,B 0,C 180,E1 -21259.886,E2 -21259.886} C_VEL
LIN {X 0,Y 206.69,Z 299.547,A -85,B 0,C 180,E1 -21264.09,E2 -21264.09} C_VEL
LIN {X 0,Y 206.688,Z 299.549,A -85,B 0,C 180,E1 -21268.437,E2 -21268.437} C_VEL
LIN {X 0,Y 206.697,Z 299.547,A -85,B 0,C 180,E1 -21272.967,E2 -21272.967} C_VEL
LIN {X 0,Y 206.673,Z 299.552,A -85,B 0,C 180,E1 -21277.751,E2 -21277.751} C_VEL
LIN {X 0,Y 206.637,Z 299.555,A -85,B 0,C 180,E1 -21281.567,E2 -21281.567} C_VEL
LIN {X 0,Y 206.638,Z 299.559,A -85,B 0,C 180,E1 -21285.591,E2 -21285.591} C_VEL
LIN {X 0,Y 206.656,Z 299.552,A -85,B 0,C 180,E1 -21289.753,E2 -21289.753} C_VEL
LIN {X 0,Y 206.713,Z 299.547,A -85,B 0,C 180,E1 -21294.696,E2 -21294.696} C_VEL
LIN {X 0,Y 206.72,Z 299.542,A -85,B 0,C 180,E1 -21299.343,E2 -21299.343} C_VEL
LIN {X 0,Y 207.346,Z 299.532,A -85,B 0,C 180,E1 -21305.405,E2 -21305.405} C_VEL
LIN {X 0,Y 207.685,Z 301.922,A -85,B 0,C 180,E1 -21306.575,E2 -21306.575} C_VEL
LIN {X 0,Y 206.277,Z 312.149,A -85,B 0,C 180,E1 -21311.569,E2 -21311.569} C_VEL
LIN {X 0,Y 206.96,Z 332.818,A -85,B 0,C 180,E1 -21312.877,E2 -21312.877} C_VEL
LIN {X 0,Y 208.671,Z 352.48,A -85,B 0,C 180,E1 -21314.059,E2 -21314.059} C_VEL
LIN {X 0,Y 208.351,Z 367.723,A -85,B 0,C 180,E1 -21315.021,E2 -21315.021} C_VEL
LIN {X 0,Y 207.656,Z 373.431,A -85,B 0,C 180,E1 -21315.39,E2 -21315.39} C_VEL
LIN {X 0,Y 204.593,Z 382.551,A -85,B 0,C 180,E1 -21316.066,E2 -21316.066} C_VEL
LIN {X 0,Y 201.447,Z 391.567,A -85,B 0,C 180,E1 -21316.858,E2 -21316.858} C_VEL
LIN {X 0,Y 200.791,Z 395.257,A -85,B 0,C 180,E1 -21317.217,E2 -21317.217} C_VEL
LIN {X 0,Y 200.717,Z 397.118,A -85,B 0,C 180,E1 -21317.409,E2 -21317.409} C_VEL
LIN {X 0,Y 200.378,Z 407.067,A -85,B 0,C 180,E1 -21318.561,E2 -21318.561} C_VEL
LIN {X 0,Y 199.952,Z 417.995,A -85,B 0,C 180,E1 -21320.2,E2 -21320.2} C_VEL
LIN {X 0,Y 199.684,Z 428.036,A -85,B 0,C 180,E1 -21322.165,E2 -21322.165} C_VEL
LIN {X 0,Y 199.472,Z 435.423,A -85,B 0,C 180,E1 -21323.936,E2 -21323.936} C_VEL
LIN {X 0,Y 199.39,Z 442.471,A -85,B 0,C 180,E1 -21325.961,E2 -21325.961} C_VEL
LIN {X 0,Y 199.19,Z 449.579,A -85,B 0,C 180,E1 -21328.487,E2 -21328.487} C_VEL
LIN {X 0,Y 198.943,Z 455.065,A -85,B 0,C 180,E1 -21331.015,E2 -21331.015} C_VEL
LIN {X 0,Y 198.368,Z 459.926,A -85,B 0,C 180,E1 -21334.067,E2 -21334.067} C_VEL
LIN {X 0,Y 198.193,Z 463.203,A -85,B 0,C 180,E1 -21336.777,E2 -21336.777} C_VEL
LIN {X 0,Y 198.275,Z 464.557,A -85,B 0,C 180,E1 -21338.154,E2 -21338.154} C_VEL
LIN {X 0,Y 199.384,Z 467.173,A -85,B 0,C 180,E1 -21342.213,E2 -21342.213} C_VEL
LIN {X 0,Y 200.496,Z 467.889,A -85,B 0,C 180,E1 -21344.207,E2 -21344.207} C_VEL
LIN {X 0,Y 201.929,Z 468.051,A -85,B 0,C 180,E1 -21346.17,E2 -21346.17} C_VEL
LIN {X 0,Y 205.75,Z 467.213,A -85,B 0,C 180,E1 -21349.976,E2 -21349.976} C_VEL
LIN {X 0,Y 208.002,Z 466.069,A -85,B 0,C 180,E1 -21351.822,E2 -21351.822} C_VEL
LIN {X 0,Y 212.189,Z 463.549,A -85,B 0,C 180,E1 -21354.461,E2 -21354.461} C_VEL
LIN {X 0,Y 216.955,Z 459.905,A -85,B 0,C 180,E1 -21356.972,E2 -21356.972} C_VEL
LIN {X 0,Y 222.342,Z 454.93,A -85,B 0,C 180,E1 -21359.34,E2 -21359.34} C_VEL
LIN {X 0,Y 227.272,Z 449.805,A -85,B 0,C 180,E1 -21361.199,E2 -21361.199} C_VEL
LIN {X 0,Y 232.546,Z 443.514,A -85,B 0,C 180,E1 -21362.959,E2 -21362.959} C_VEL
LIN {X 0,Y 238.382,Z 435.696,A -85,B 0,C 180,E1 -21364.632,E2 -21364.632} C_VEL
LIN {X 0,Y 244.824,Z 425.659,A -85,B 0,C 180,E1 -21366.242,E2 -21366.242} C_VEL
LIN {X 0,Y 249.483,Z 417.06,A -85,B 0,C 180,E1 -21367.279,E2 -21367.279} C_VEL
LIN {X 0,Y 255.179,Z 404.795,A -85,B 0,C 180,E1 -21368.407,E2 -21368.407} C_VEL
LIN {X 0,Y 259.294,Z 393.428,A -85,B 0,C 180,E1 -21369.189,E2 -21369.189} C_VEL
LIN {X 0,Y 262.141,Z 383.501,A -85,B 0,C 180,E1 -21369.73,E2 -21369.73} C_VEL
LIN {X 0,Y 261.725,Z 380.157,A -85,B 0,C 180,E1 -21371.401,E2 -21371.401} C_VEL
LIN {X 0,Y 261.334,Z 377.248,A -85,B 0,C 180,E1 -21373.759,E2 -21373.759} C_VEL
LIN {X 0,Y 261.248,Z 376.503,A -85,B 0,C 180,E1 -21375.61,E2 -21375.61} C_VEL
LIN {X 0,Y 261.641,Z 376.686,A -85,B 0,C 180,E1 -21377.807,E2 -21377.807} C_VEL
LIN {X 0,Y 262.551,Z 378.272,A -85,B 0,C 180,E1 -21380.091,E2 -21380.091} C_VEL
LIN {X 0,Y 262.853,Z 379.251,A -85,B 0,C 180,E1 -21380.747,E2 -21380.747} C_VEL
LIN {X 0,Y 260.107,Z 389.05,A -85,B 0,C 180,E1 -21381.335,E2 -21381.335} C_VEL
LIN {X 0,Y 256.788,Z 398.436,A -85,B 0,C 180,E1 -21382.032,E2 -21382.032} C_VEL
LIN {X 0,Y 251.946,Z 409.531,A -85,B 0,C 180,E1 -21383.141,E2 -21383.141} C_VEL
LIN {X 0,Y 247.121,Z 418.742,A -85,B 0,C 180,E1 -21384.33,E2 -21384.33} C_VEL
LIN {X 0,Y 241.45,Z 427.998,A -85,B 0,C 180,E1 -21385.914,E2 -21385.914} C_VEL
LIN {X 0,Y 234.91,Z 436.72,A -85,B 0,C 180,E1 -21387.916,E2 -21387.916} C_VEL
LIN {X 0,Y 229.753,Z 442.616,A -85,B 0,C 180,E1 -21389.679,E2 -21389.679} C_VEL
LIN {X 0,Y 225.894,Z 446.466,A -85,B 0,C 180,E1 -21391.16,E2 -21391.16} C_VEL
LIN {X 0,Y 220.544,Z 451.101,A -85,B 0,C 180,E1 -21393.496,E2 -21393.496} C_VEL
LIN {X 0,Y 217.239,Z 453.472,A -85,B 0,C 180,E1 -21395.121,E2 -21395.121} C_VEL
LIN {X 0,Y 214.115,Z 455.358,A -85,B 0,C 180,E1 -21396.795,E2 -21396.795} C_VEL
LIN {X 0,Y 211.263,Z 456.745,A -85,B 0,C 180,E1 -21398.526,E2 -21398.526} C_VEL
LIN {X 0,Y 208.645,Z 457.575,A -85,B 0,C 180,E1 -21400.306,E2 -21400.306} C_VEL
LIN {X 0,Y 206.251,Z 457.959,A -85,B 0,C 180,E1 -21402.132,E2 -21402.132} C_VEL
LIN {X 0,Y 204.183,Z 457.928,A -85,B 0,C 180,E1 -21404.007,E2 -21404.007} C_VEL
LIN {X 0,Y 202.553,Z 457.41,A -85,B 0,C 180,E1 -21405.934,E2 -21405.934} C_VEL
LIN {X 0,Y 200.968,Z 456.342,A -85,B 0,C 180,E1 -21407.878,E2 -21407.878} C_VEL
LIN {X 0,Y 199.268,Z 453.873,A -85,B 0,C 180,E1 -21410.96,E2 -21410.96} C_VEL
LIN {X 0,Y 198.4,Z 450.52,A -85,B 0,C 180,E1 -21413.89,E2 -21413.89} C_VEL
LIN {X 0,Y 197.98,Z 445.733,A -85,B 0,C 180,E1 -21416.938,E2 -21416.938} C_VEL
LIN {X 0,Y 197.95,Z 439.475,A -85,B 0,C 180,E1 -21419.99,E2 -21419.99} C_VEL
LIN {X 0,Y 198.279,Z 433.028,A -85,B 0,C 180,E1 -21422.529,E2 -21422.529} C_VEL
LIN {X 0,Y 198.414,Z 426.648,A -85,B 0,C 180,E1 -21424.561,E2 -21424.561} C_VEL
LIN {X 0,Y 198.851,Z 418.344,A -85,B 0,C 180,E1 -21426.765,E2 -21426.765} C_VEL
LIN {X 0,Y 199.311,Z 407.936,A -85,B 0,C 180,E1 -21428.937,E2 -21428.937} C_VEL
LIN {X 0,Y 199.84,Z 397.785,A -85,B 0,C 180,E1 -21430.629,E2 -21430.629} C_VEL
LIN {X 0,Y 200.357,Z 384.81,A -85,B 0,C 180,E1 -21432.267,E2 -21432.267} C_VEL
LIN {X 0,Y 200.783,Z 373.772,A -85,B 0,C 180,E1 -21433.269,E2 -21433.269} C_VEL
LIN {X 0,Y 201.855,Z 320.489,A -85,B 0,C 180,E1 -21436.779,E2 -21436.779} C_VEL
LIN {X 0,Y 199.806,Z 300.411,A -85,B 0,C 180,E1 -21438.04,E2 -21438.04} C_VEL
LIN {X 0,Y 199.703,Z 300.416,A -85,B 0,C 180,E1 -21442.763,E2 -21442.763} C_VEL
LIN {X 0,Y 199.652,Z 300.428,A -85,B 0,C 180,E1 -21448.348,E2 -21448.348} C_VEL
LIN {X 0,Y 199.65,Z 300.425,A -85,B 0,C 180,E1 -21452.34,E2 -21452.34} C_VEL
LIN {X 0,Y 199.597,Z 300.435,A -85,B 0,C 180,E1 -21456.754,E2 -21456.754} C_VEL
LIN {X 0,Y 199.573,Z 300.433,A -85,B 0,C 180,E1 -21459.321,E2 -21459.321} C_VEL
LIN {X 0,Y 199.542,Z 300.438,A -85,B 0,C 180,E1 -21462.296,E2 -21462.296} C_VEL
LIN {X 0,Y 199.552,Z 300.44,A -85,B 0,C 180,E1 -21465.217,E2 -21465.217} C_VEL
LIN {X 0,Y 199.547,Z 300.437,A -85,B 0,C 180,E1 -21467.993,E2 -21467.993} C_VEL
LIN {X 0,Y 199.569,Z 300.435,A -85,B 0,C 180,E1 -21470.762,E2 -21470.762} C_VEL
LIN {X 0,Y 199.578,Z 300.435,A -85,B 0,C 180,E1 -21475.703,E2 -21475.703} C_VEL
LIN {X 0,Y 199.652,Z 300.422,A -85,B 0,C 180,E1 -21478.125,E2 -21478.125} C_VEL
LIN {X 0,Y 199.642,Z 300.428,A -85,B 0,C 180,E1 -21482.762,E2 -21482.762} C_VEL
LIN {X 0,Y 199.675,Z 300.422,A -85,B 0,C 180,E1 -21487.218,E2 -21487.218} C_VEL
LIN {X 0,Y 199.755,Z 300.415,A -85,B 0,C 180,E1 -21491.752,E2 -21491.752} C_VEL
LIN {X 0,Y 199.785,Z 300.407,A -85,B 0,C 180,E1 -21495.741,E2 -21495.741} C_VEL
LIN {X 0,Y 200.008,Z 300.385,A -85,B 0,C 180,E1 -21499.878,E2 -21499.878} C_VEL
LIN {X 0,Y 199.983,Z 300.384,A -85,B 0,C 180,E1 -21503.945,E2 -21503.945} C_VEL
LIN {X 0,Y 200.301,Z 300.347,A -85,B 0,C 180,E1 -21507.986,E2 -21507.986} C_VEL
LIN {X 0,Y 200.437,Z 300.332,A -85,B 0,C 180,E1 -21509.997,E2 -21509.997} C_VEL
LIN {X 0,Y 200.3,Z 300.347,A -85,B 0,C 180,E1 -21512.007,E2 -21512.007} C_VEL
LIN {X 0,Y 200.049,Z 300.379,A -85,B 0,C 180,E1 -21518.075,E2 -21518.075} C_VEL
LIN {X 0,Y 199.83,Z 300.405,A -85,B 0,C 180,E1 -21522.178,E2 -21522.178} C_VEL
LIN {X 0,Y 199.747,Z 300.416,A -85,B 0,C 180,E1 -21526.344,E2 -21526.344} C_VEL
LIN {X 0,Y 199.632,Z 300.429,A -85,B 0,C 180,E1 -21530.609,E2 -21530.609} C_VEL
LIN {X 0,Y 199.617,Z 300.432,A -85,B 0,C 180,E1 -21534.988,E2 -21534.988} C_VEL
LIN {X 0,Y 199.629,Z 300.427,A -85,B 0,C 180,E1 -21539.525,E2 -21539.525} C_VEL
LIN {X 0,Y 199.618,Z 300.427,A -85,B 0,C 180,E1 -21542.355,E2 -21542.355} C_VEL
LIN {X 0,Y 199.61,Z 300.433,A -85,B 0,C 180,E1 -21546.761,E2 -21546.761} C_VEL
LIN {X 0,Y 199.659,Z 300.423,A -85,B 0,C 180,E1 -21549.311,E2 -21549.311} C_VEL
LIN {X 0,Y 199.649,Z 300.425,A -85,B 0,C 180,E1 -21552.352,E2 -21552.352} C_VEL
LIN {X 0,Y 199.654,Z 300.429,A -85,B 0,C 180,E1 -21555.267,E2 -21555.267} C_VEL
LIN {X 0,Y 199.64,Z 300.425,A -85,B 0,C 180,E1 -21558.037,E2 -21558.037} C_VEL
LIN {X 0,Y 199.643,Z 300.424,A -85,B 0,C 180,E1 -21560.75,E2 -21560.75} C_VEL
LIN {X 0,Y 199.598,Z 300.434,A -85,B 0,C 180,E1 -21565.725,E2 -21565.725} C_VEL
LIN {X 0,Y 199.662,Z 300.421,A -85,B 0,C 180,E1 -21568.144,E2 -21568.144} C_VEL
LIN {X 0,Y 199.654,Z 300.426,A -85,B 0,C 180,E1 -21572.78,E2 -21572.78} C_VEL
LIN {X 0,Y 199.683,Z 300.419,A -85,B 0,C 180,E1 -21577.235,E2 -21577.235} C_VEL
LIN {X 0,Y 199.724,Z 300.419,A -85,B 0,C 180,E1 -21581.808,E2 -21581.808} C_VEL
LIN {X 0,Y 199.791,Z 300.408,A -85,B 0,C 180,E1 -21585.756,E2 -21585.756} C_VEL
LIN {X 0,Y 200.002,Z 300.383,A -85,B 0,C 180,E1 -21589.892,E2 -21589.892} C_VEL
LIN {X 0,Y 199.99,Z 300.384,A -85,B 0,C 180,E1 -21593.959,E2 -21593.959} C_VEL
LIN {X 0,Y 200.274,Z 300.348,A -85,B 0,C 180,E1 -21597.999,E2 -21597.999} C_VEL
LIN {X 0,Y 200.433,Z 300.33,A -85,B 0,C 180,E1 -21600.01,E2 -21600.01} C_VEL
LIN {X 0,Y 199.985,Z 300.382,A -85,B 0,C 180,E1 -21604.04,E2 -21604.04} C_VEL
LIN {X 0,Y 200.06,Z 300.375,A -85,B 0,C 180,E1 -21608.088,E2 -21608.088} C_VEL
LIN {X 0,Y 199.848,Z 300.4,A -85,B 0,C 180,E1 -21612.191,E2 -21612.191} C_VEL
LIN {X 0,Y 199.736,Z 300.415,A -85,B 0,C 180,E1 -21616.359,E2 -21616.359} C_VEL
LIN {X 0,Y 199.638,Z 300.428,A -85,B 0,C 180,E1 -21620.622,E2 -21620.622} C_VEL
LIN {X 0,Y 199.62,Z 300.431,A -85,B 0,C 180,E1 -21625.001,E2 -21625.001} C_VEL
LIN {X 0,Y 199.609,Z 300.431,A -85,B 0,C 180,E1 -21629.543,E2 -21629.543} C_VEL
LIN {X 0,Y 199.668,Z 300.421,A -85,B 0,C 180,E1 -21632.361,E2 -21632.361} C_VEL
LIN {X 0,Y 199.622,Z 300.43,A -85,B 0,C 180,E1 -21636.774,E2 -21636.774} C_VEL
LIN {X 0,Y 199.601,Z 300.433,A -85,B 0,C 180,E1 -21639.34,E2 -21639.34} C_VEL
LIN {X 0,Y 199.573,Z 300.435,A -85,B 0,C 180,E1 -21642.315,E2 -21642.315} C_VEL
LIN {X 0,Y 199.584,Z 300.435,A -85,B 0,C 180,E1 -21645.235,E2 -21645.235} C_VEL
LIN {X 0,Y 199.579,Z 300.434,A -85,B 0,C 180,E1 -21648.01,E2 -21648.01} C_VEL
LIN {X 0,Y 199.608,Z 300.429,A -85,B 0,C 180,E1 -21650.781,E2 -21650.781} C_VEL
LIN {X 0,Y 199.624,Z 300.431,A -85,B 0,C 180,E1 -21655.72,E2 -21655.72} C_VEL
LIN {X 0,Y 199.699,Z 300.419,A -85,B 0,C 180,E1 -21658.141,E2 -21658.141} C_VEL
LIN {X 0,Y 200.406,Z 300.363,A -85,B 0,C 180,E1 -21665.771,E2 -21665.771} C_VEL
LIN {X 0,Y 200.365,Z 303.405,A -85,B 0,C 180,E1 -21667.308,E2 -21667.308} C_VEL
LIN {X 0,Y 199.203,Z 311.964,A -85,B 0,C 180,E1 -21671.663,E2 -21671.663} C_VEL
LIN {X 0,Y 199.898,Z 333.009,A -85,B 0,C 180,E1 -21673.032,E2 -21673.032} C_VEL
LIN {X 0,Y 201.614,Z 352.776,A -85,B 0,C 180,E1 -21674.265,E2 -21674.265} C_VEL
LIN {X 0,Y 200.865,Z 391.954,A -85,B 0,C 180,E1 -21676.922,E2 -21676.922} C_VEL
LIN {X 0,Y 200.717,Z 397.118,A -85,B 0,C 180,E1 -21677.409,E2 -21677.409} C_VEL
LIN {X 0,Y 200.245,Z 400.764,A -85,B 0,C 180,E1 -21677.805,E2 -21677.805} C_VEL
LIN {X 0,Y 198.756,Z 405.933,A -85,B 0,C 180,E1 -21678.516,E2 -21678.516} C_VEL
LIN {X 0,Y 193.713,Z 417.934,A -85,B 0,C 180,E1 -21680.684,E2 -21680.684} C_VEL
LIN {X 0,Y 192.88,Z 423.653,A -85,B 0,C 180,E1 -21681.84,E2 -21681.84} C_VEL
LIN {X 0,Y 192.666,Z 431.947,A -85,B 0,C 180,E1 -21683.721,E2 -21683.721} C_VEL
LIN {X 0,Y 192.578,Z 439.479,A -85,B 0,C 180,E1 -21685.818,E2 -21685.818} C_VEL
LIN {X 0,Y 192.454,Z 445.588,A -85,B 0,C 180,E1 -21687.911,E2 -21687.911} C_VEL
LIN {X 0,Y 192.288,Z 451.743,A -85,B 0,C 180,E1 -21690.527,E2 -21690.527} C_VEL
LIN {X 0,Y 191.707,Z 456.497,A -85,B 0,C 180,E1 -21693.156,E2 -21693.156} C_VEL
LIN {X 0,Y 191.385,Z 459.599,A -85,B 0,C 180,E1 -21695.271,E2 -21695.271} C_VEL
LIN {X 0,Y 191.394,Z 463.125,A -85,B 0,C 180,E1 -21698.45,E2 -21698.45} C_VEL
LIN {X 0,Y 191.743,Z 464.937,A -85,B 0,C 180,E1 -21700.564,E2 -21700.564} C_VEL
LIN {X 0,Y 192.514,Z 466.278,A -85,B 0,C 180,E1 -21702.656,E2 -21702.656} C_VEL
LIN {X 0,Y 195.143,Z 467.578,A -85,B 0,C 180,E1 -21706.749,E2 -21706.749} C_VEL
LIN {X 0,Y 196.932,Z 467.654,A -85,B 0,C 180,E1 -21708.738,E2 -21708.738} C_VEL
LIN {X 0,Y 201.433,Z 466.322,A -85,B 0,C 180,E1 -21712.572,E2 -21712.572} C_VEL
LIN {X 0,Y 204.244,Z 465.087,A -85,B 0,C 180,E1 -21714.391,E2 -21714.391} C_VEL
LIN {X 0,Y 208.992,Z 462.222,A -85,B 0,C 180,E1 -21717.002,E2 -21717.002} C_VEL
LIN {X 0,Y 214.388,Z 458.255,A -85,B 0,C 180,E1 -21719.457,E2 -21719.457} C_VEL
LIN {X 0,Y 220.336,Z 453.03,A -85,B 0,C 180,E1 -21721.759,E2 -21721.759} C_VEL
LIN {X 0,Y 226.828,Z 446.433,A -85,B 0,C 180,E1 -21723.901,E2 -21723.901} C_VEL
LIN {X 0,Y 232.702,Z 439.559,A -85,B 0,C 180,E1 -21725.551,E2 -21725.551} C_VEL
LIN {X 0,Y 238.636,Z 431.395,A -85,B 0,C 180,E1 -21727.025,E2 -21727.025} C_VEL
LIN {X 0,Y 244.139,Z 422.842,A -85,B 0,C 180,E1 -21728.24,E2 -21728.24} C_VEL
LIN {X 0,Y 249.621,Z 412.936,A -85,B 0,C 180,E1 -21729.31,E2 -21729.31} C_VEL
LIN {X 0,Y 255.103,Z 400.509,A -85,B 0,C 180,E1 -21730.296,E2 -21730.296} C_VEL
LIN {X 0,Y 259.46,Z 388.29,A -85,B 0,C 180,E1 -21731.043,E2 -21731.043} C_VEL
LIN {X 0,Y 259.474,Z 386.649,A -85,B 0,C 180,E1 -21731.793,E2 -21731.793} C_VEL
LIN {X 0,Y 259.304,Z 383.879,A -85,B 0,C 180,E1 -21734.088,E2 -21734.088} C_VEL
LIN {X 0,Y 259.239,Z 383.383,A -85,B 0,C 180,E1 -21735.174,E2 -21735.174} C_VEL
LIN {X 0,Y 259.54,Z 383.351,A -85,B 0,C 180,E1 -21737.385,E2 -21737.385} C_VEL
LIN {X 0,Y 260.112,Z 384.273,A -85,B 0,C 180,E1 -21739.163,E2 -21739.163} C_VEL
LIN {X 0,Y 259.942,Z 385.541,A -85,B 0,C 180,E1 -21739.535,E2 -21739.535} C_VEL
LIN {X 0,Y 255.827,Z 397.054,A -85,B 0,C 180,E1 -21740.32,E2 -21740.32} C_VEL
LIN {X 0,Y 251.341,Z 407.479,A -85,B 0,C 180,E1 -21741.262,E2 -21741.262} C_VEL
LIN {X 0,Y 245.597,Z 418.128,A -85,B 0,C 180,E1 -21742.541,E2 -21742.541} C_VEL
LIN {X 0,Y 240.738,Z 425.702,A -85,B 0,C 180,E1 -21743.752,E2 -21743.752} C_VEL
LIN {X 0,Y 234.881,Z 433.725,A -85,B 0,C 180,E1 -21745.345,E2 -21745.345} C_VEL
LIN {X 0,Y 228.201,Z 441.311,A -85,B 0,C 180,E1 -21747.379,E2 -21747.379} C_VEL
LIN {X 0,Y 221.924,Z 447.232,A -85,B 0,C 180,E1 -21749.547,E2 -21749.547} C_VEL
LIN {X 0,Y 216.188,Z 451.771,A -85,B 0,C 180,E1 -21751.867,E2 -21751.867} C_VEL
LIN {X 0,Y 210.964,Z 455.067,A -85,B 0,C 180,E1 -21754.328,E2 -21754.328} C_VEL
LIN {X 0,Y 207.037,Z 456.898,A -85,B 0,C 180,E1 -21756.43,E2 -21756.43} C_VEL
LIN {X 0,Y 202.025,Z 458.299,A -85,B 0,C 180,E1 -21759.633,E2 -21759.633} C_VEL
LIN {X 0,Y 199.521,Z 458.431,A -85,B 0,C 180,E1 -21761.508,E2 -21761.508} C_VEL
LIN {X 0,Y 197.389,Z 458.049,A -85,B 0,C 180,E1 -21763.441,E2 -21763.441} C_VEL
LIN {X 0,Y 195.675,Z 457.276,A -85,B 0,C 180,E1 -21765.429,E2 -21765.429} C_VEL
LIN {X 0,Y 194.05,Z 456.086,A -85,B 0,C 180,E1 -21767.439,E2 -21767.439} C_VEL
LIN {X 0,Y 192.201,Z 452.895,A -85,B 0,C 180,E1 -21770.868,E2 -21770.868} C_VEL
LIN {X 0,Y 191.448,Z 449.388,A -85,B 0,C 180,E1 -21773.667,E2 -21773.667} C_VEL
LIN {X 0,Y 191.148,Z 446.189,A -85,B 0,C 180,E1 -21775.773,E2 -21775.773} C_VEL
LIN {X 0,Y 190.992,Z 440.011,A -85,B 0,C 180,E1 -21778.935,E2 -21778.935} C_VEL
LIN {X 0,Y 191.248,Z 433.613,A -85,B 0,C 180,E1 -21781.569,E2 -21781.569} C_VEL
LIN {X 0,Y 191.439,Z 427.391,A -85,B 0,C 180,E1 -21783.673,E2 -21783.673} C_VEL
LIN {X 0,Y 191.87,Z 418,A -85,B 0,C 180,E1 -21786.298,E2 -21786.298} C_VEL
LIN {X 0,Y 192.317,Z 408.341,A -85,B 0,C 180,E1 -21788.394,E2 -21788.394} C_VEL
LIN {X 0,Y 192.848,Z 397.521,A -85,B 0,C 180,E1 -21790.259,E2 -21790.259} C_VEL
LIN {X 0,Y 193.295,Z 385.885,A -85,B 0,C 180,E1 -21791.79,E2 -21791.79} C_VEL
LIN {X 0,Y 193.775,Z 374.389,A -85,B 0,C 180,E1 -21792.89,E2 -21792.89} C_VEL
LIN {X 0,Y 194.74,Z 320.609,A -85,B 0,C 180,E1 -21796.634,E2 -21796.634} C_VEL
LIN {X 0,Y 192.766,Z 301.289,A -85,B 0,C 180,E1 -21797.91,E2 -21797.91} C_VEL
LIN {X 0,Y 192.666,Z 301.293,A -85,B 0,C 180,E1 -21803.644,E2 -21803.644} C_VEL
LIN {X 0,Y 192.588,Z 301.305,A -85,B 0,C 180,E1 -21808.853,E2 -21808.853} C_VEL
LIN {X 0,Y 192.579,Z 301.306,A -85,B 0,C 180,E1 -21813.175,E2 -21813.175} C_VEL
LIN {X 0,Y 192.521,Z 301.316,A -85,B 0,C 180,E1 -21818.343,E2 -21818.343} C_VEL
LIN {X 0,Y 192.461,Z 301.323,A -85,B 0,C 180,E1 -21823.082,E2 -21823.082} C_VEL
LIN {X 0,Y 192.461,Z 301.323,A -85,B 0,C 180,E1 -21826.895,E2 -21826.895} C_VEL
LIN {X 0,Y 192.513,Z 301.315,A -85,B 0,C 180,E1 -21831.635,E2 -21831.635} C_VEL
LIN {X 0,Y 192.562,Z 301.31,A -85,B 0,C 180,E1 -21836.803,E2 -21836.803} C_VEL
LIN {X 0,Y 192.618,Z 301.303,A -85,B 0,C 180,E1 -21841.681,E2 -21841.681} C_VEL
LIN {X 0,Y 192.647,Z 301.296,A -85,B 0,C 180,E1 -21846.337,E2 -21846.337} C_VEL
LIN {X 0,Y 192.691,Z 301.296,A -85,B 0,C 180,E1 -21851.452,E2 -21851.452} C_VEL
